LIN {X 0,Y 349.192,Z 815.635,A -85,B 0,C 180,E1 16408.843,E2 16408.843} C_VEL
LIN {X 0,Y 352.149,Z 828.309,A -85,B 0,C 180,E1 16411.517,E2 16411.517} C_VEL
LIN {X 0,Y 338.548,Z 866.043,A -85,B 0,C 180,E1 16414.618,E2 16414.618} C_VEL
LIN {X 0,Y 323.279,Z 901.225,A -85,B 0,C 180,E1 16418.786,E2 16418.786} C_VEL
LIN {X 0,Y 308.073,Z 932.384,A -85,B 0,C 180,E1 16424.048,E2 16424.048} C_VEL
LIN {X 0,Y 293.775,Z 959.9,A -85,B 0,C 180,E1 16430.633,E2 16430.633} C_VEL
LIN {X 0,Y 281.914,Z 983.359,A -85,B 0,C 180,E1 16438.716,E2 16438.716} C_VEL
LIN {X 0,Y 274.605,Z 1000.274,A -85,B 0,C 180,E1 16447.297,E2 16447.297} C_VEL
LIN {X 0,Y 271.389,Z 1010.786,A -85,B 0,C 180,E1 16455.461,E2 16455.461} C_VEL
LIN {X 0,Y 270.341,Z 1016.72,A -85,B 0,C 180,E1 16463.569,E2 16463.569} C_VEL
LIN {X 0,Y 270.547,Z 1018.167,A -85,B 0,C 180,E1 16470.001,E2 16470.001} C_VEL
LIN {X 0,Y 270.343,Z 1016.724,A -85,B 0,C 180,E1 16476.432,E2 16476.432} C_VEL
LIN {X 0,Y 271.389,Z 1010.794,A -85,B 0,C 180,E1 16484.541,E2 16484.541} C_VEL
LIN {X 0,Y 274.599,Z 1000.292,A -85,B 0,C 180,E1 16492.704,E2 16492.704} C_VEL
LIN {X 0,Y 281.856,Z 983.603,A -85,B 0,C 180,E1 16501.184,E2 16501.184} C_VEL
LIN {X 0,Y 293.699,Z 960.03,A -85,B 0,C 180,E1 16509.349,E2 16509.349} C_VEL
LIN {X 0,Y 308.953,Z 930.715,A -85,B 0,C 180,E1 16516.291,E2 16516.291} C_VEL
LIN {X 0,Y 325.073,Z 897.549,A -85,B 0,C 180,E1 16521.735,E2 16521.735} C_VEL
LIN {X 0,Y 340.684,Z 860.965,A -85,B 0,C 180,E1 16525.883,E2 16525.883} C_VEL
LIN {X 0,Y 350.17,Z 834.984,A -85,B 0,C 180,E1 16528.014,E2 16528.014} C_VEL
LIN {X 0,Y 350.059,Z 829.98,A -85,B 0,C 180,E1 16528.799,E2 16528.799} C_VEL
LIN {X 0,Y 345.076,Z 822.989,A -85,B 0,C 180,E1 16531.277,E2 16531.277} C_VEL
LIN {X 0,Y 338.35,Z 801.661,A -85,B 0,C 180,E1 16536.945,E2 16536.945} C_VEL
LIN {X 0,Y 331.725,Z 785.413,A -85,B 0,C 180,E1 16542.789,E2 16542.789} C_VEL
LIN {X 0,Y 326.179,Z 773.809,A -85,B 0,C 180,E1 16549.075,E2 16549.075} C_VEL
LIN {X 0,Y 323.36,Z 767.768,A -85,B 0,C 180,E1 16554.2,E2 16554.2} C_VEL
LIN {X 0,Y 321.912,Z 765.9,A -85,B 0,C 180,E1 16561.341,E2 16561.341} C_VEL
LIN {X 0,Y 323.589,Z 768.974,A -85,B 0,C 180,E1 16567.85,E2 16567.85} C_VEL
LIN {X 0,Y 326.59,Z 776.623,A -85,B 0,C 180,E1 16573.395,E2 16573.395} C_VEL
LIN {X 0,Y 332.226,Z 790.347,A -85,B 0,C 180,E1 16579.977,E2 16579.977} C_VEL
LIN {X 0,Y 338.405,Z 808.971,A -85,B 0,C 180,E1 16586.141,E2 16586.141} C_VEL
LIN {X 0,Y 342.983,Z 830.452,A -85,B 0,C 180,E1 16591.603,E2 16591.603} C_VEL
LIN {X 0,Y 342.674,Z 834.152,A -85,B 0,C 180,E1 16592.188,E2 16592.188} C_VEL
LIN {X 0,Y 326.849,Z 872.233,A -85,B 0,C 180,E1 16596.121,E2 16596.121} C_VEL
LIN {X 0,Y 310.06,Z 906.091,A -85,B 0,C 180,E1 16601.239,E2 16601.239} C_VEL
LIN {X 0,Y 294.191,Z 934.724,A -85,B 0,C 180,E1 16607.507,E2 16607.507} C_VEL
LIN {X 0,Y 279.881,Z 959.338,A -85,B 0,C 180,E1 16615.387,E2 16615.387} C_VEL
LIN {X 0,Y 269.909,Z 977.851,A -85,B 0,C 180,E1 16624.312,E2 16624.312} C_VEL
LIN {X 0,Y 264.694,Z 989.892,A -85,B 0,C 180,E1 16633.38,E2 16633.38} C_VEL
LIN {X 0,Y 263.017,Z 995.241,A -85,B 0,C 180,E1 16640.055,E2 16640.055} C_VEL
LIN {X 0,Y 262.515,Z 997.859,A -85,B 0,C 180,E1 16646.693,E2 16646.693} C_VEL
LIN {X 0,Y 262.472,Z 997.841,A -85,B 0,C 180,E1 16653.306,E2 16653.306} C_VEL
LIN {X 0,Y 263.46,Z 993.471,A -85,B 0,C 180,E1 16662.392,E2 16662.392} C_VEL
LIN {X 0,Y 266.708,Z 984.794,A -85,B 0,C 180,E1 16670.856,E2 16670.856} C_VEL
LIN {X 0,Y 273.935,Z 969.98,A -85,B 0,C 180,E1 16679.83,E2 16679.83} C_VEL
LIN {X 0,Y 285.315,Z 950.061,A -85,B 0,C 180,E1 16687.828,E2 16687.828} C_VEL
LIN {X 0,Y 300.025,Z 924.248,A -85,B 0,C 180,E1 16694.951,E2 16694.951} C_VEL
LIN {X 0,Y 316.458,Z 893.504,A -85,B 0,C 180,E1 16700.788,E2 16700.788} C_VEL
LIN {X 0,Y 332.912,Z 858.489,A -85,B 0,C 180,E1 16705.349,E2 16705.349} C_VEL
LIN {X 0,Y 343.162,Z 831.415,A -85,B 0,C 180,E1 16708.043,E2 16708.043} C_VEL
LIN {X 0,Y 338.289,Z 809.145,A -85,B 0,C 180,E1 16713.727,E2 16713.727} C_VEL
LIN {X 0,Y 332.65,Z 791.782,A -85,B 0,C 180,E1 16719.354,E2 16719.354} C_VEL
LIN {X 0,Y 327.088,Z 777.911,A -85,B 0,C 180,E1 16725.66,E2 16725.66} C_VEL
LIN {X 0,Y 323.78,Z 770.112,A -85,B 0,C 180,E1 16731.102,E2 16731.102} C_VEL
LIN {X 0,Y 322.787,Z 767.547,A -85,B 0,C 180,E1 16733.611,E2 16733.611} C_VEL
LIN {X 0,Y 321.875,Z 765.702,A -85,B 0,C 180,E1 16741.27,E2 16741.27} C_VEL
LIN {X 0,Y 324.017,Z 769.137,A -85,B 0,C 180,E1 16747.557,E2 16747.557} C_VEL
LIN {X 0,Y 327.173,Z 775.881,A -85,B 0,C 180,E1 16752.389,E2 16752.389} C_VEL
LIN {X 0,Y 332.03,Z 786.449,A -85,B 0,C 180,E1 16757.658,E2 16757.658} C_VEL
LIN {X 0,Y 338.631,Z 802.667,A -85,B 0,C 180,E1 16763.383,E2 16763.383} C_VEL
LIN {X 0,Y 345.418,Z 824.473,A -85,B 0,C 180,E1 16769.104,E2 16769.104} C_VEL
LIN {X 0,Y 346.743,Z 831.868,A -85,B 0,C 180,E1 16770.654,E2 16770.654} C_VEL
LIN {X 0,Y 332.245,Z 869.964,A -85,B 0,C 180,E1 16773.902,E2 16773.902} C_VEL
LIN {X 0,Y 316.574,Z 904.239,A -85,B 0,C 180,E1 16778.125,E2 16778.125} C_VEL
LIN {X 0,Y 301.211,Z 934.227,A -85,B 0,C 180,E1 16783.38,E2 16783.38} C_VEL
LIN {X 0,Y 286.56,Z 961.124,A -85,B 0,C 180,E1 16790.048,E2 16790.048} C_VEL
LIN {X 0,Y 274.435,Z 983.878,A -85,B 0,C 180,E1 16798.193,E2 16798.193} C_VEL
LIN {X 0,Y 266.586,Z 1001.235,A -85,B 0,C 180,E1 16807.458,E2 16807.458} C_VEL
LIN {X 0,Y 263.22,Z 1012.101,A -85,B 0,C 180,E1 16816.698,E2 16816.698} C_VEL
LIN {X 0,Y 262.434,Z 1016.421,A -85,B 0,C 180,E1 16823.375,E2 16823.375} C_VEL
LIN {X 0,Y 262.646,Z 1017.87,A -85,B 0,C 180,E1 16830.001,E2 16830.001} C_VEL
LIN {X 0,Y 262.437,Z 1016.426,A -85,B 0,C 180,E1 16836.627,E2 16836.627} C_VEL
LIN {X 0,Y 263.59,Z 1010.492,A -85,B 0,C 180,E1 16844.981,E2 16844.981} C_VEL
LIN {X 0,Y 267.06,Z 999.986,A -85,B 0,C 180,E1 16853.383,E2 16853.383} C_VEL
LIN {X 0,Y 275.011,Z 982.798,A -85,B 0,C 180,E1 16862.297,E2 16862.297} C_VEL
LIN {X 0,Y 287.357,Z 959.722,A -85,B 0,C 180,E1 16870.394,E2 16870.394} C_VEL
LIN {X 0,Y 302.879,Z 931.245,A -85,B 0,C 180,E1 16877.258,E2 16877.258} C_VEL
LIN {X 0,Y 319.89,Z 897.653,A -85,B 0,C 180,E1 16882.83,E2 16882.83} C_VEL
LIN {X 0,Y 335.722,Z 861.9,A -85,B 0,C 180,E1 16886.915,E2 16886.915} C_VEL
LIN {X 0,Y 346.968,Z 830.772,A -85,B 0,C 180,E1 16889.492,E2 16889.492} C_VEL
LIN {X 0,Y 345.076,Z 822.989,A -85,B 0,C 180,E1 16891.277,E2 16891.277} C_VEL
LIN {X 0,Y 341.723,Z 817.584,A -85,B 0,C 180,E1 16893.191,E2 16893.191} C_VEL
LIN {X 0,Y 335.269,Z 810.574,A -85,B 0,C 180,E1 16896.583,E2 16896.583} C_VEL
LIN {X 0,Y 329.616,Z 795.321,A -85,B 0,C 180,E1 16901.933,E2 16901.933} C_VEL
LIN {X 0,Y 324.144,Z 782.486,A -85,B 0,C 180,E1 16908.343,E2 16908.343} C_VEL
LIN {X 0,Y 320.93,Z 775.179,A -85,B 0,C 180,E1 16914.58,E2 16914.58} C_VEL
LIN {X 0,Y 319.755,Z 773.301,A -85,B 0,C 180,E1 16919.993,E2 16919.993} C_VEL
LIN {X 0,Y 320.822,Z 775.397,A -85,B 0,C 180,E1 16926.77,E2 16926.77} C_VEL
LIN {X 0,Y 324.466,Z 785.539,A -85,B 0,C 180,E1 16934.172,E2 16934.172} C_VEL
LIN {X 0,Y 329.739,Z 800.223,A -85,B 0,C 180,E1 16940.836,E2 16940.836} C_VEL
LIN {X 0,Y 334.912,Z 819.087,A -85,B 0,C 180,E1 16946.866,E2 16946.866} C_VEL
LIN {X 0,Y 337.643,Z 836.643,A -85,B 0,C 180,E1 16951.23,E2 16951.23} C_VEL
LIN {X 0,Y 321.513,Z 873.886,A -85,B 0,C 180,E1 16955.138,E2 16955.138} C_VEL
LIN {X 0,Y 304.044,Z 907.647,A -85,B 0,C 180,E1 16960.328,E2 16960.328} C_VEL
LIN {X 0,Y 287.404,Z 936.344,A -85,B 0,C 180,E1 16966.775,E2 16966.775} C_VEL
LIN {X 0,Y 273.19,Z 959.643,A -85,B 0,C 180,E1 16974.412,E2 16974.412} C_VEL
LIN {X 0,Y 262.601,Z 978.179,A -85,B 0,C 180,E1 16983.56,E2 16983.56} C_VEL
LIN {X 0,Y 257.012,Z 990.192,A -85,B 0,C 180,E1 16992.868,E2 16992.868} C_VEL
LIN {X 0,Y 255.16,Z 995.54,A -85,B 0,C 180,E1 16999.745,E2 16999.745} C_VEL
LIN {X 0,Y 254.63,Z 998.155,A -85,B 0,C 180,E1 17006.59,E2 17006.59} C_VEL
LIN {X 0,Y 254.59,Z 998.137,A -85,B 0,C 180,E1 17013.409,E2 17013.409} C_VEL
LIN {X 0,Y 255.559,Z 994.036,A -85,B 0,C 180,E1 17022.386,E2 17022.386} C_VEL
LIN {X 0,Y 259.115,Z 985.194,A -85,B 0,C 180,E1 17031.42,E2 17031.42} C_VEL
LIN {X 0,Y 266.883,Z 970.287,A -85,B 0,C 180,E1 17040.702,E2 17040.702} C_VEL
LIN {X 0,Y 279.288,Z 949.73,A -85,B 0,C 180,E1 17049.065,E2 17049.065} C_VEL
LIN {X 0,Y 294.334,Z 924.555,A -85,B 0,C 180,E1 17056.068,E2 17056.068} C_VEL
LIN {X 0,Y 311.165,Z 894.279,A -85,B 0,C 180,E1 17061.87,E2 17061.87} C_VEL
LIN {X 0,Y 327.828,Z 860.177,A -85,B 0,C 180,E1 17066.356,E2 17066.356} C_VEL
LIN {X 0,Y 337.792,Z 836.164,A -85,B 0,C 180,E1 17068.696,E2 17068.696} C_VEL
LIN {X 0,Y 334.138,Z 816.442,A -85,B 0,C 180,E1 17073.793,E2 17073.793} C_VEL
LIN {X 0,Y 328.985,Z 798.23,A -85,B 0,C 180,E1 17079.817,E2 17079.817} C_VEL
LIN {X 0,Y 323.83,Z 784.12,A -85,B 0,C 180,E1 17086.489,E2 17086.489} C_VEL
LIN {X 0,Y 320.962,Z 776.22,A -85,B 0,C 180,E1 17092.15,E2 17092.15} C_VEL
LIN {X 0,Y 319.624,Z 772.942,A -85,B 0,C 180,E1 17100.007,E2 17100.007} C_VEL
LIN {X 0,Y 321.547,Z 776.325,A -85,B 0,C 180,E1 17107.191,E2 17107.191} C_VEL
LIN {X 0,Y 326.002,Z 786.606,A -85,B 0,C 180,E1 17114.186,E2 17114.186} C_VEL
LIN {X 0,Y 332.256,Z 801.967,A -85,B 0,C 180,E1 17120.685,E2 17120.685} C_VEL
LIN {X 0,Y 338.803,Z 822.716,A -85,B 0,C 180,E1 17126.808,E2 17126.808} C_VEL
LIN {X 0,Y 341.672,Z 834.738,A -85,B 0,C 180,E1 17129.722,E2 17129.722} C_VEL
LIN {X 0,Y 325.744,Z 874.43,A -85,B 0,C 180,E1 17133.213,E2 17133.213} C_VEL
LIN {X 0,Y 308.657,Z 909.78,A -85,B 0,C 180,E1 17137.817,E2 17137.817} C_VEL
LIN {X 0,Y 291.346,Z 941.598,A -85,B 0,C 180,E1 17143.895,E2 17143.895} C_VEL
LIN {X 0,Y 275.826,Z 968.396,A -85,B 0,C 180,E1 17151.362,E2 17151.362} C_VEL
LIN {X 0,Y 264.539,Z 989.281,A -85,B 0,C 180,E1 17159.947,E2 17159.947} C_VEL
LIN {X 0,Y 257.678,Z 1004.486,A -85,B 0,C 180,E1 17169.357,E2 17169.357} C_VEL
LIN {X 0,Y 255.097,Z 1012.945,A -85,B 0,C 180,E1 17177.832,E2 17177.832} C_VEL
LIN {X 0,Y 254.608,Z 1017.208,A -85,B 0,C 180,E1 17186.591,E2 17186.591} C_VEL
LIN {X 0,Y 254.548,Z 1017.208,A -85,B 0,C 180,E1 17193.411,E2 17193.411} C_VEL
LIN {X 0,Y 255.108,Z 1012.946,A -85,B 0,C 180,E1 17202.181,E2 17202.181} C_VEL
LIN {X 0,Y 257.652,Z 1004.502,A -85,B 0,C 180,E1 17210.646,E2 17210.646} C_VEL
LIN {X 0,Y 264.538,Z 989.306,A -85,B 0,C 180,E1 17220.054,E2 17220.054} C_VEL
LIN {X 0,Y 276.522,Z 967.268,A -85,B 0,C 180,E1 17229.027,E2 17229.027} C_VEL
LIN {X 0,Y 292.299,Z 939.965,A -85,B 0,C 180,E1 17236.485,E2 17236.485} C_VEL
LIN {X 0,Y 309.624,Z 908.014,A -85,B 0,C 180,E1 17242.458,E2 17242.458} C_VEL
LIN {X 0,Y 326.654,Z 872.547,A -85,B 0,C 180,E1 17246.99,E2 17246.99} C_VEL
LIN {X 0,Y 341.581,Z 834.062,A -85,B 0,C 180,E1 17250.452,E2 17250.452} C_VEL
LIN {X 0,Y 335.818,Z 812.344,A -85,B 0,C 180,E1 17256.057,E2 17256.057} C_VEL
LIN {X 0,Y 335.269,Z 810.574,A -85,B 0,C 180,E1 17256.583,E2 17256.583} C_VEL
LIN {X 0,Y 331.982,Z 806.597,A -85,B 0,C 180,E1 17258.657,E2 17258.657} C_VEL
LIN {X 0,Y 326.134,Z 802.071,A -85,B 0,C 180,E1 17262.299,E2 17262.299} C_VEL
LIN {X 0,Y 321.4,Z 790.016,A -85,B 0,C 180,E1 17268.446,E2 17268.446} C_VEL
LIN {X 0,Y 318.386,Z 782.743,A -85,B 0,C 180,E1 17274.536,E2 17274.536} C_VEL
LIN {X 0,Y 317.226,Z 780.794,A -85,B 0,C 180,E1 17279.993,E2 17279.993} C_VEL
LIN {X 0,Y 318.241,Z 783.088,A -85,B 0,C 180,E1 17286.825,E2 17286.825} C_VEL
LIN {X 0,Y 321.541,Z 793.293,A -85,B 0,C 180,E1 17294.304,E2 17294.304} C_VEL
LIN {X 0,Y 326.297,Z 808.189,A -85,B 0,C 180,E1 17300.984,E2 17300.984} C_VEL
LIN {X 0,Y 330.606,Z 826.564,A -85,B 0,C 180,E1 17306.877,E2 17306.877} C_VEL
LIN {X 0,Y 332.243,Z 840.085,A -85,B 0,C 180,E1 17310.333,E2 17310.333} C_VEL
LIN {X 0,Y 316.498,Z 875.047,A -85,B 0,C 180,E1 17314.059,E2 17314.059} C_VEL
LIN {X 0,Y 298.871,Z 907.947,A -85,B 0,C 180,E1 17319.146,E2 17319.146} C_VEL
LIN {X 0,Y 281.49,Z 936.649,A -85,B 0,C 180,E1 17325.633,E2 17325.633} C_VEL
LIN {X 0,Y 266.334,Z 960.267,A -85,B 0,C 180,E1 17333.519,E2 17333.519} C_VEL
LIN {X 0,Y 255.33,Z 978.522,A -85,B 0,C 180,E1 17342.775,E2 17342.775} C_VEL
LIN {X 0,Y 249.319,Z 990.494,A -85,B 0,C 180,E1 17352.323,E2 17352.323} C_VEL
LIN {X 0,Y 247.312,Z 995.839,A -85,B 0,C 180,E1 17359.416,E2 17359.416} C_VEL
LIN {X 0,Y 246.725,Z 998.452,A -85,B 0,C 180,E1 17366.481,E2 17366.481} C_VEL
LIN {X 0,Y 246.685,Z 998.434,A -85,B 0,C 180,E1 17373.518,E2 17373.518} C_VEL
LIN {X 0,Y 247.568,Z 994.868,A -85,B 0,C 180,E1 17381.972,E2 17381.972} C_VEL
LIN {X 0,Y 251.095,Z 986.61,A -85,B 0,C 180,E1 17391.21,E2 17391.21} C_VEL
LIN {X 0,Y 258.948,Z 972.277,A -85,B 0,C 180,E1 17400.771,E2 17400.771} C_VEL
LIN {X 0,Y 272.273,Z 951.216,A -85,B 0,C 180,E1 17409.754,E2 17409.754} C_VEL
LIN {X 0,Y 288.749,Z 924.863,A -85,B 0,C 180,E1 17417.231,E2 17417.231} C_VEL
LIN {X 0,Y 306.107,Z 894.856,A -85,B 0,C 180,E1 17423.016,E2 17423.016} C_VEL
LIN {X 0,Y 323.791,Z 859.668,A -85,B 0,C 180,E1 17427.629,E2 17427.629} C_VEL
LIN {X 0,Y 332.434,Z 838.872,A -85,B 0,C 180,E1 17429.739,E2 17429.739} C_VEL
LIN {X 0,Y 328.718,Z 818.125,A -85,B 0,C 180,E1 17435.52,E2 17435.52} C_VEL
LIN {X 0,Y 324.28,Z 801.901,A -85,B 0,C 180,E1 17441.394,E2 17441.394} C_VEL
LIN {X 0,Y 320.216,Z 789.549,A -85,B 0,C 180,E1 17447.723,E2 17447.723} C_VEL
LIN {X 0,Y 318.024,Z 783.165,A -85,B 0,C 180,E1 17453.035,E2 17453.035} C_VEL
LIN {X 0,Y 317.101,Z 780.442,A -85,B 0,C 180,E1 17460.007,E2 17460.007} C_VEL
LIN {X 0,Y 318.933,Z 784.119,A -85,B 0,C 180,E1 17467.25,E2 17467.25} C_VEL
LIN {X 0,Y 322.662,Z 793.144,A -85,B 0,C 180,E1 17473.574,E2 17473.574} C_VEL
LIN {X 0,Y 328.407,Z 808.289,A -85,B 0,C 180,E1 17480.21,E2 17480.21} C_VEL
LIN {X 0,Y 334.045,Z 828.023,A -85,B 0,C 180,E1 17486.229,E2 17486.229} C_VEL
LIN {X 0,Y 336.04,Z 838.94,A -85,B 0,C 180,E1 17488.871,E2 17488.871} C_VEL
LIN {X 0,Y 320.665,Z 875.582,A -85,B 0,C 180,E1 17492.162,E2 17492.162} C_VEL
LIN {X 0,Y 302.655,Z 911.323,A -85,B 0,C 180,E1 17496.896,E2 17496.896} C_VEL
LIN {X 0,Y 285.213,Z 942.034,A -85,B 0,C 180,E1 17502.881,E2 17502.881} C_VEL
LIN {X 0,Y 269.365,Z 968.165,A -85,B 0,C 180,E1 17510.293,E2 17510.293} C_VEL
LIN {X 0,Y 257.431,Z 988.97,A -85,B 0,C 180,E1 17519.028,E2 17519.028} C_VEL
LIN {X 0,Y 250.048,Z 1004.179,A -85,B 0,C 180,E1 17528.697,E2 17528.697} C_VEL
LIN {X 0,Y 247.248,Z 1012.646,A -85,B 0,C 180,E1 17537.442,E2 17537.442} C_VEL
LIN {X 0,Y 246.693,Z 1016.91,A -85,B 0,C 180,E1 17546.482,E2 17546.482} C_VEL
LIN {X 0,Y 246.636,Z 1016.911,A -85,B 0,C 180,E1 17553.52,E2 17553.52} C_VEL
LIN {X 0,Y 247.241,Z 1012.764,A -85,B 0,C 180,E1 17562.406,E2 17562.406} C_VEL
LIN {X 0,Y 250.024,Z 1004.197,A -85,B 0,C 180,E1 17571.306,E2 17571.306} C_VEL
LIN {X 0,Y 257.442,Z 988.998,A -85,B 0,C 180,E1 17580.972,E2 17580.972} C_VEL
LIN {X 0,Y 270.046,Z 967.123,A -85,B 0,C 180,E1 17590.08,E2 17590.08} C_VEL
LIN {X 0,Y 286.663,Z 939.657,A -85,B 0,C 180,E1 17597.685,E2 17597.685} C_VEL
LIN {X 0,Y 304.478,Z 908.171,A -85,B 0,C 180,E1 17603.607,E2 17603.607} C_VEL
LIN {X 0,Y 322.231,Z 872.422,A -85,B 0,C 180,E1 17608.182,E2 17608.182} C_VEL
LIN {X 0,Y 336.284,Z 837.943,A -85,B 0,C 180,E1 17611.286,E2 17611.286} C_VEL
LIN {X 0,Y 331.082,Z 816.695,A -85,B 0,C 180,E1 17617.051,E2 17617.051} C_VEL
LIN {X 0,Y 326.134,Z 802.071,A -85,B 0,C 180,E1 17622.299,E2 17622.299} C_VEL
LIN {X 0,Y 323.169,Z 799.664,A -85,B 0,C 180,E1 17624.521,E2 17624.521} C_VEL
LIN {X 0,Y 318.665,Z 798.307,A -85,B 0,C 180,E1 17627.991,E2 17627.991} C_VEL
LIN {X 0,Y 318.417,Z 797.734,A -85,B 0,C 180,E1 17628.374,E2 17628.374} C_VEL
LIN {X 0,Y 315.746,Z 790.323,A -85,B 0,C 180,E1 17634.491,E2 17634.491} C_VEL
LIN {X 0,Y 314.656,Z 788.271,A -85,B 0,C 180,E1 17639.993,E2 17639.993} C_VEL
LIN {X 0,Y 315.442,Z 790.714,A -85,B 0,C 180,E1 17646.884,E2 17646.884} C_VEL
LIN {X 0,Y 318.445,Z 801.039,A -85,B 0,C 180,E1 17654.408,E2 17654.408} C_VEL
LIN {X 0,Y 322.289,Z 814.685,A -85,B 0,C 180,E1 17660.619,E2 17660.619} C_VEL
LIN {X 0,Y 325.89,Z 832.625,A -85,B 0,C 180,E1 17666.516,E2 17666.516} C_VEL
LIN {X 0,Y 327.024,Z 843.334,A -85,B 0,C 180,E1 17669.394,E2 17669.394} C_VEL
LIN {X 0,Y 310.953,Z 877.44,A -85,B 0,C 180,E1 17673.109,E2 17673.109} C_VEL
LIN {X 0,Y 293.385,Z 908.928,A -85,B 0,C 180,E1 17678.047,E2 17678.047} C_VEL
LIN {X 0,Y 275.757,Z 936.95,A -85,B 0,C 180,E1 17684.456,E2 17684.456} C_VEL
LIN {X 0,Y 259.6,Z 960.887,A -85,B 0,C 180,E1 17692.587,E2 17692.587} C_VEL
LIN {X 0,Y 248.467,Z 978.3,A -85,B 0,C 180,E1 17701.556,E2 17701.556} C_VEL
LIN {X 0,Y 241.674,Z 990.794,A -85,B 0,C 180,E1 17711.744,E2 17711.744} C_VEL
LIN {X 0,Y 239.503,Z 996.137,A -85,B 0,C 180,E1 17719.067,E2 17719.067} C_VEL
LIN {X 0,Y 238.819,Z 998.749,A -85,B 0,C 180,E1 17726.364,E2 17726.364} C_VEL
LIN {X 0,Y 238.78,Z 998.731,A -85,B 0,C 180,E1 17733.635,E2 17733.635} C_VEL
LIN {X 0,Y 239.749,Z 995.168,A -85,B 0,C 180,E1 17742.369,E2 17742.369} C_VEL
LIN {X 0,Y 243.563,Z 986.915,A -85,B 0,C 180,E1 17751.899,E2 17751.899} C_VEL
LIN {X 0,Y 251.96,Z 972.585,A -85,B 0,C 180,E1 17761.722,E2 17761.722} C_VEL
LIN {X 0,Y 266.018,Z 951.526,A -85,B 0,C 180,E1 17770.884,E2 17770.884} C_VEL
LIN {X 0,Y 283.284,Z 925.172,A -85,B 0,C 180,E1 17778.44,E2 17778.44} C_VEL
LIN {X 0,Y 301.613,Z 894.615,A -85,B 0,C 180,E1 17784.328,E2 17784.328} C_VEL
LIN {X 0,Y 319.425,Z 860.312,A -85,B 0,C 180,E1 17788.806,E2 17788.806} C_VEL
LIN {X 0,Y 327.031,Z 842.333,A -85,B 0,C 180,E1 17790.694,E2 17790.694} C_VEL
LIN {X 0,Y 323.919,Z 822.212,A -85,B 0,C 180,E1 17796.6,E2 17796.6} C_VEL
LIN {X 0,Y 320.013,Z 806.768,A -85,B 0,C 180,E1 17802.563,E2 17802.563} C_VEL
LIN {X 0,Y 316.592,Z 795.336,A -85,B 0,C 180,E1 17808.98,E2 17808.98} C_VEL
LIN {X 0,Y 314.85,Z 789.72,A -85,B 0,C 180,E1 17814.488,E2 17814.488} C_VEL
LIN {X 0,Y 314.55,Z 787.914,A -85,B 0,C 180,E1 17820.007,E2 17820.007} C_VEL
LIN {X 0,Y 316.081,Z 791.293,A -85,B 0,C 180,E1 17826.884,E2 17826.884} C_VEL
LIN {X 0,Y 319.714,Z 800.938,A -85,B 0,C 180,E1 17833.702,E2 17833.702} C_VEL
LIN {X 0,Y 324.614,Z 815.273,A -85,B 0,C 180,E1 17839.99,E2 17839.99} C_VEL
LIN {X 0,Y 329.514,Z 834.289,A -85,B 0,C 180,E1 17845.885,E2 17845.885} C_VEL
LIN {X 0,Y 330.722,Z 842.44,A -85,B 0,C 180,E1 17847.94,E2 17847.94} C_VEL
LIN {X 0,Y 314.941,Z 878.272,A -85,B 0,C 180,E1 17851.254,E2 17851.254} C_VEL
LIN {X 0,Y 297.03,Z 912.353,A -85,B 0,C 180,E1 17855.857,E2 17855.857} C_VEL
LIN {X 0,Y 279.127,Z 942.546,A -85,B 0,C 180,E1 17861.842,E2 17861.842} C_VEL
LIN {X 0,Y 263.218,Z 967.625,A -85,B 0,C 180,E1 17869.061,E2 17869.061} C_VEL
LIN {X 0,Y 249.941,Z 989.378,A -85,B 0,C 180,E1 17878.455,E2 17878.455} C_VEL
LIN {X 0,Y 242.482,Z 1003.873,A -85,B 0,C 180,E1 17887.998,E2 17887.998} C_VEL
LIN {X 0,Y 239.379,Z 1012.472,A -85,B 0,C 180,E1 17897.211,E2 17897.211} C_VEL
LIN {X 0,Y 238.777,Z 1016.613,A -85,B 0,C 180,E1 17906.365,E2 17906.365} C_VEL
LIN {X 0,Y 238.997,Z 1016.983,A -85,B 0,C 180,E1 17910.001,E2 17910.001} C_VEL
LIN {X 0,Y 238.774,Z 1015.533,A -85,B 0,C 180,E1 17917.287,E2 17917.287} C_VEL
LIN {X 0,Y 240.244,Z 1009.585,A -85,B 0,C 180,E1 17926.476,E2 17926.476} C_VEL
LIN {X 0,Y 245.178,Z 998.055,A -85,B 0,C 180,E1 17936.336,E2 17936.336} C_VEL
LIN {X 0,Y 254.591,Z 981.512,A -85,B 0,C 180,E1 17945.44,E2 17945.44} C_VEL
LIN {X 0,Y 269.509,Z 957.981,A -85,B 0,C 180,E1 17954.046,E2 17954.046} C_VEL
LIN {X 0,Y 286.972,Z 929.845,A -85,B 0,C 180,E1 17960.979,E2 17960.979} C_VEL
LIN {X 0,Y 305.496,Z 897.168,A -85,B 0,C 180,E1 17966.435,E2 17966.435} C_VEL
LIN {X 0,Y 323.506,Z 860.096,A -85,B 0,C 180,E1 17970.603,E2 17970.603} C_VEL
LIN {X 0,Y 330.943,Z 841.734,A -85,B 0,C 180,E1 17972.176,E2 17972.176} C_VEL
LIN {X 0,Y 326.758,Z 822.529,A -85,B 0,C 180,E1 17977.594,E2 17977.594} C_VEL
LIN {X 0,Y 321.803,Z 806.64,A -85,B 0,C 180,E1 17983.598,E2 17983.598} C_VEL
LIN {X 0,Y 318.417,Z 797.734,A -85,B 0,C 180,E1 17988.374,E2 17988.374} C_VEL
LIN {X 0,Y 316.353,Z 796.484,A -85,B 0,C 180,E1 17990.69,E2 17990.69} C_VEL
LIN {X 0,Y 312.754,Z 797.678,A -85,B 0,C 180,E1 17994.678,E2 17994.678} C_VEL
LIN {X 0,Y 311.787,Z 795.642,A -85,B 0,C 180,E1 17999.993,E2 17999.993} C_VEL
LIN {X 0,Y 312.513,Z 798.292,A -85,B 0,C 180,E1 18006.949,E2 18006.949} C_VEL
LIN {X 0,Y 314.834,Z 807.547,A -85,B 0,C 180,E1 18013.905,E2 18013.905} C_VEL
LIN {X 0,Y 318.27,Z 821.612,A -85,B 0,C 180,E1 18020.435,E2 18020.435} C_VEL
LIN {X 0,Y 321.02,Z 837.659,A -85,B 0,C 180,E1 18025.855,E2 18025.855} C_VEL
LIN {X 0,Y 321.768,Z 846.913,A -85,B 0,C 180,E1 18028.46,E2 18028.46} C_VEL
LIN {X 0,Y 303.775,Z 883.088,A -85,B 0,C 180,E1 18032.566,E2 18032.566} C_VEL
LIN {X 0,Y 285.136,Z 914.538,A -85,B 0,C 180,E1 18037.826,E2 18037.826} C_VEL
LIN {X 0,Y 267.542,Z 940.913,A -85,B 0,C 180,E1 18044.29,E2 18044.29} C_VEL
LIN {X 0,Y 251.815,Z 963.069,A -85,B 0,C 180,E1 18052.301,E2 18052.301} C_VEL
LIN {X 0,Y 240.86,Z 979.29,A -85,B 0,C 180,E1 18061.117,E2 18061.117} C_VEL
LIN {X 0,Y 234.028,Z 991.096,A -85,B 0,C 180,E1 18071.126,E2 18071.126} C_VEL
LIN {X 0,Y 231.664,Z 996.436,A -85,B 0,C 180,E1 18078.692,E2 18078.692} C_VEL
LIN {X 0,Y 230.914,Z 999.046,A -85,B 0,C 180,E1 18086.24,E2 18086.24} C_VEL
LIN {X 0,Y 230.875,Z 999.029,A -85,B 0,C 180,E1 18093.759,E2 18093.759} C_VEL
LIN {X 0,Y 232.041,Z 995.219,A -85,B 0,C 180,E1 18103.199,E2 18103.199} C_VEL
LIN {X 0,Y 236.06,Z 987.22,A -85,B 0,C 180,E1 18112.633,E2 18112.633} C_VEL
LIN {X 0,Y 245.081,Z 972.891,A -85,B 0,C 180,E1 18122.721,E2 18122.721} C_VEL
LIN {X 0,Y 259.881,Z 951.835,A -85,B 0,C 180,E1 18132.066,E2 18132.066} C_VEL
LIN {X 0,Y 277.974,Z 925.478,A -85,B 0,C 180,E1 18139.689,E2 18139.689} C_VEL
LIN {X 0,Y 296.701,Z 895.391,A -85,B 0,C 180,E1 18145.525,E2 18145.525} C_VEL
LIN {X 0,Y 315.527,Z 860.249,A -85,B 0,C 180,E1 18150.087,E2 18150.087} C_VEL
LIN {X 0,Y 321.778,Z 846.533,A -85,B 0,C 180,E1 18151.484,E2 18151.484} C_VEL
LIN {X 0,Y 319.361,Z 827.786,A -85,B 0,C 180,E1 18157.197,E2 18157.197} C_VEL
LIN {X 0,Y 316.073,Z 812.545,A -85,B 0,C 180,E1 18163.346,E2 18163.346} C_VEL
LIN {X 0,Y 313.505,Z 802.924,A -85,B 0,C 180,E1 18168.87,E2 18168.87} C_VEL
LIN {X 0,Y 311.981,Z 797.125,A -85,B 0,C 180,E1 18174.437,E2 18174.437} C_VEL
LIN {X 0,Y 311.69,Z 795.265,A -85,B 0,C 180,E1 18180.007,E2 18180.007} C_VEL
LIN {X 0,Y 313.153,Z 798.871,A -85,B 0,C 180,E1 18186.948,E2 18186.948} C_VEL
LIN {X 0,Y 316.552,Z 808.715,A -85,B 0,C 180,E1 18193.841,E2 18193.841} C_VEL
LIN {X 0,Y 321.024,Z 823.438,A -85,B 0,C 180,E1 18200.223,E2 18200.223} C_VEL
LIN {X 0,Y 325.257,Z 843.257,A -85,B 0,C 180,E1 18206.338,E2 18206.338} C_VEL
LIN {X 0,Y 325.147,Z 846.868,A -85,B 0,C 180,E1 18207.056,E2 18207.056} C_VEL
LIN {X 0,Y 307.223,Z 885.137,A -85,B 0,C 180,E1 18210.789,E2 18210.789} C_VEL
LIN {X 0,Y 287.573,Z 920.096,A -85,B 0,C 180,E1 18215.921,E2 18215.921} C_VEL
LIN {X 0,Y 268.015,Z 950.844,A -85,B 0,C 180,E1 18222.744,E2 18222.744} C_VEL
LIN {X 0,Y 252.275,Z 974.556,A -85,B 0,C 180,E1 18230.6,E2 18230.6} C_VEL
LIN {X 0,Y 239.665,Z 994.572,A -85,B 0,C 180,E1 18240.669,E2 18240.669} C_VEL
LIN {X 0,Y 233.183,Z 1007.612,A -85,B 0,C 180,E1 18251.056,E2 18251.056} C_VEL
LIN {X 0,Y 231.216,Z 1013.684,A -85,B 0,C 180,E1 18259.196,E2 18259.196} C_VEL
LIN {X 0,Y 230.862,Z 1016.315,A -85,B 0,C 180,E1 18266.24,E2 18266.24} C_VEL
LIN {X 0,Y 231.094,Z 1016.687,A -85,B 0,C 180,E1 18270.001,E2 18270.001} C_VEL
LIN {X 0,Y 230.87,Z 1015.234,A -85,B 0,C 180,E1 18277.538,E2 18277.538} C_VEL
LIN {X 0,Y 232.504,Z 1009.282,A -85,B 0,C 180,E1 18287.041,E2 18287.041} C_VEL
LIN {X 0,Y 237.564,Z 998.303,A -85,B 0,C 180,E1 18296.836,E2 18296.836} C_VEL
LIN {X 0,Y 247.91,Z 981.204,A -85,B 0,C 180,E1 18306.547,E2 18306.547} C_VEL
LIN {X 0,Y 263.579,Z 957.67,A -85,B 0,C 180,E1 18315.306,E2 18315.306} C_VEL
LIN {X 0,Y 282.245,Z 928.954,A -85,B 0,C 180,E1 18322.386,E2 18322.386} C_VEL
LIN {X 0,Y 301.71,Z 895.704,A -85,B 0,C 180,E1 18327.871,E2 18327.871} C_VEL
LIN {X 0,Y 319.57,Z 859.865,A -85,B 0,C 180,E1 18331.865,E2 18331.865} C_VEL
LIN {X 0,Y 325.572,Z 844.966,A -85,B 0,C 180,E1 18333.248,E2 18333.248} C_VEL
LIN {X 0,Y 321.509,Z 824.984,A -85,B 0,C 180,E1 18339.259,E2 18339.259} C_VEL
LIN {X 0,Y 317.068,Z 810.228,A -85,B 0,C 180,E1 18345.476,E2 18345.476} C_VEL
LIN {X 0,Y 313.68,Z 800.94,A -85,B 0,C 180,E1 18351.668,E2 18351.668} C_VEL
LIN {X 0,Y 312.754,Z 797.678,A -85,B 0,C 180,E1 18354.678,E2 18354.678} C_VEL
LIN {X 0,Y 310.524,Z 799.884,A -85,B 0,C 180,E1 18357.834,E2 18357.834} C_VEL
LIN {X 0,Y 308.724,Z 803.184,A -85,B 0,C 180,E1 18361.031,E2 18361.031} C_VEL
LIN {X 0,Y 309.335,Z 805.751,A -85,B 0,C 180,E1 18367.021,E2 18367.021} C_VEL
LIN {X 0,Y 311.402,Z 815.214,A -85,B 0,C 180,E1 18374.061,E2 18374.061} C_VEL
LIN {X 0,Y 314.185,Z 828.907,A -85,B 0,C 180,E1 18380.44,E2 18380.44} C_VEL
LIN {X 0,Y 316.173,Z 844.803,A -85,B 0,C 180,E1 18385.851,E2 18385.851} C_VEL
LIN {X 0,Y 316.266,Z 851.098,A -85,B 0,C 180,E1 18387.563,E2 18387.563} C_VEL
LIN {X 0,Y 298.116,Z 885.934,A -85,B 0,C 180,E1 18391.615,E2 18391.615} C_VEL
LIN {X 0,Y 278.627,Z 917.35,A -85,B 0,C 180,E1 18397.018,E2 18397.018} C_VEL
LIN {X 0,Y 259.555,Z 944.57,A -85,B 0,C 180,E1 18404.024,E2 18404.024} C_VEL
LIN {X 0,Y 243.16,Z 966.57,A -85,B 0,C 180,E1 18412.62,E2 18412.62} C_VEL
LIN {X 0,Y 231.364,Z 983.142,A -85,B 0,C 180,E1 18422.735,E2 18422.735} C_VEL
LIN {X 0,Y 225.569,Z 992.917,A -85,B 0,C 180,E1 18432.418,E2 18432.418} C_VEL
LIN {X 0,Y 223.185,Z 998.374,A -85,B 0,C 180,E1 18442.201,E2 18442.201} C_VEL
LIN {X 0,Y 223.148,Z 999.652,A -85,B 0,C 180,E1 18449.999,E2 18449.999} C_VEL
LIN {X 0,Y 223.157,Z 998.338,A -85,B 0,C 180,E1 18457.798,E2 18457.798} C_VEL
LIN {X 0,Y 225.585,Z 992.833,A -85,B 0,C 180,E1 18467.579,E2 18467.579} C_VEL
LIN {X 0,Y 231.411,Z 982.998,A -85,B 0,C 180,E1 18477.257,E2 18477.257} C_VEL
LIN {X 0,Y 243.259,Z 966.37,A -85,B 0,C 180,E1 18487.36,E2 18487.36} C_VEL
LIN {X 0,Y 260.061,Z 943.735,A -85,B 0,C 180,E1 18496.12,E2 18496.12} C_VEL
LIN {X 0,Y 279.032,Z 916.571,A -85,B 0,C 180,E1 18503.031,E2 18503.031} C_VEL
LIN {X 0,Y 298.454,Z 885.205,A -85,B 0,C 180,E1 18508.37,E2 18508.37} C_VEL
LIN {X 0,Y 316.482,Z 849.634,A -85,B 0,C 180,E1 18512.614,E2 18512.614} C_VEL
LIN {X 0,Y 314.353,Z 830.435,A -85,B 0,C 180,E1 18518.834,E2 18518.834} C_VEL
LIN {X 0,Y 311.505,Z 816.208,A -85,B 0,C 180,E1 18525.224,E2 18525.224} C_VEL
LIN {X 0,Y 309.401,Z 807.017,A -85,B 0,C 180,E1 18531.566,E2 18531.566} C_VEL
LIN {X 0,Y 308.597,Z 803.269,A -85,B 0,C 180,E1 18537.195,E2 18537.195} C_VEL
LIN {X 0,Y 308.776,Z 802.609,A -85,B 0,C 180,E1 18540.007,E2 18540.007} C_VEL
LIN {X 0,Y 309.969,Z 805.876,A -85,B 0,C 180,E1 18546.572,E2 18546.572} C_VEL
LIN {X 0,Y 312.87,Z 815.151,A -85,B 0,C 180,E1 18553.321,E2 18553.321} C_VEL
LIN {X 0,Y 316.631,Z 829.026,A -85,B 0,C 180,E1 18559.56,E2 18559.56} C_VEL
LIN {X 0,Y 320.153,Z 847.535,A -85,B 0,C 180,E1 18565.499,E2 18565.499} C_VEL
LIN {X 0,Y 319.427,Z 851.382,A -85,B 0,C 180,E1 18566.173,E2 18566.173} C_VEL
LIN {X 0,Y 301.882,Z 887.105,A -85,B 0,C 180,E1 18569.742,E2 18569.742} C_VEL
LIN {X 0,Y 282.415,Z 920.432,A -85,B 0,C 180,E1 18574.694,E2 18574.694} C_VEL
LIN {X 0,Y 262.512,Z 950.534,A -85,B 0,C 180,E1 18581.428,E2 18581.428} C_VEL
LIN {X 0,Y 245.461,Z 974.863,A -85,B 0,C 180,E1 18589.634,E2 18589.634} C_VEL
LIN {X 0,Y 232.506,Z 994.284,A -85,B 0,C 180,E1 18599.691,E2 18599.691} C_VEL
LIN {X 0,Y 225.498,Z 1007.306,A -85,B 0,C 180,E1 18610.384,E2 18610.384} C_VEL
LIN {X 0,Y 223.409,Z 1013.123,A -85,B 0,C 180,E1 18618.27,E2 18618.27} C_VEL
LIN {X 0,Y 222.967,Z 1016.018,A -85,B 0,C 180,E1 18626.107,E2 18626.107} C_VEL
LIN {X 0,Y 223.19,Z 1016.391,A -85,B 0,C 180,E1 18630.001,E2 18630.001} C_VEL
LIN {X 0,Y 222.981,Z 1014.936,A -85,B 0,C 180,E1 18637.806,E2 18637.806} C_VEL
LIN {X 0,Y 224.773,Z 1008.979,A -85,B 0,C 180,E1 18647.646,E2 18647.646} C_VEL
LIN {X 0,Y 229.991,Z 998.453,A -85,B 0,C 180,E1 18657.441,E2 18657.441} C_VEL
LIN {X 0,Y 241.331,Z 980.896,A -85,B 0,C 180,E1 18667.714,E2 18667.714} C_VEL
LIN {X 0,Y 257.751,Z 957.458,A -85,B 0,C 180,E1 18676.587,E2 18676.587} C_VEL
LIN {X 0,Y 276.759,Z 929.538,A -85,B 0,C 180,E1 18683.555,E2 18683.555} C_VEL
LIN {X 0,Y 297.127,Z 896.004,A -85,B 0,C 180,E1 18689.123,E2 18689.123} C_VEL
LIN {X 0,Y 315.822,Z 859.599,A -85,B 0,C 180,E1 18693.156,E2 18693.156} C_VEL
LIN {X 0,Y 320.355,Z 848.66,A -85,B 0,C 180,E1 18694.213,E2 18694.213} C_VEL
LIN {X 0,Y 317.203,Z 831.018,A -85,B 0,C 180,E1 18699.749,E2 18699.749} C_VEL
LIN {X 0,Y 313.334,Z 816.625,A -85,B 0,C 180,E1 18706.014,E2 18706.014} C_VEL
LIN {X 0,Y 310.545,Z 808.382,A -85,B 0,C 180,E1 18711.584,E2 18711.584} C_VEL
LIN {X 0,Y 309.684,Z 805.046,A -85,B 0,C 180,E1 18714.774,E2 18714.774} C_VEL
LIN {X 0,Y 308.724,Z 803.184,A -85,B 0,C 180,E1 18721.031,E2 18721.031} C_VEL
LIN {X 0,Y 307.794,Z 805.979,A -85,B 0,C 180,E1 18723.401,E2 18723.401} C_VEL
LIN {X 0,Y 306.081,Z 813.398,A -85,B 0,C 180,E1 18727.287,E2 18727.287} C_VEL
LIN {X 0,Y 307.496,Z 821.402,A -85,B 0,C 180,E1 18733.445,E2 18733.445} C_VEL
LIN {X 0,Y 309.628,Z 833.858,A -85,B 0,C 180,E1 18739.549,E2 18739.549} C_VEL
LIN {X 0,Y 311.218,Z 850.267,A -85,B 0,C 180,E1 18745.346,E2 18745.346} C_VEL
LIN {X 0,Y 310.764,Z 855.145,A -85,B 0,C 180,E1 18746.631,E2 18746.631} C_VEL
LIN {X 0,Y 292.849,Z 888.044,A -85,B 0,C 180,E1 18750.539,E2 18750.539} C_VEL
LIN {X 0,Y 272.185,Z 919.934,A -85,B 0,C 180,E1 18756.159,E2 18756.159} C_VEL
LIN {X 0,Y 253.386,Z 945.623,A -85,B 0,C 180,E1 18762.946,E2 18762.946} C_VEL
LIN {X 0,Y 236.693,Z 966.874,A -85,B 0,C 180,E1 18771.413,E2 18771.413} C_VEL
LIN {X 0,Y 224.185,Z 983.445,A -85,B 0,C 180,E1 18781.786,E2 18781.786} C_VEL
LIN {X 0,Y 217.905,Z 993.218,A -85,B 0,C 180,E1 18791.779,E2 18791.779} C_VEL
LIN {X 0,Y 215.309,Z 998.672,A -85,B 0,C 180,E1 18801.914,E2 18801.914} C_VEL
LIN {X 0,Y 215.247,Z 999.949,A -85,B 0,C 180,E1 18809.999,E2 18809.999} C_VEL
LIN {X 0,Y 215.692,Z 997.554,A -85,B 0,C 180,E1 18820.752,E2 18820.752} C_VEL
LIN {X 0,Y 218.853,Z 991.599,A -85,B 0,C 180,E1 18830.237,E2 18830.237} C_VEL
LIN {X 0,Y 227.184,Z 979.265,A -85,B 0,C 180,E1 18841.225,E2 18841.225} C_VEL
LIN {X 0,Y 241.364,Z 960.974,A -85,B 0,C 180,E1 18851.192,E2 18851.192} C_VEL
LIN {X 0,Y 260.251,Z 936.407,A -85,B 0,C 180,E1 18859.712,E2 18859.712} C_VEL
LIN {X 0,Y 280.292,Z 907.888,A -85,B 0,C 180,E1 18866.152,E2 18866.152} C_VEL
LIN {X 0,Y 301.143,Z 873.495,A -85,B 0,C 180,E1 18871.258,E2 18871.258} C_VEL
LIN {X 0,Y 310.809,Z 854.783,A -85,B 0,C 180,E1 18873.302,E2 18873.302} C_VEL
LIN {X 0,Y 310.383,Z 841.273,A -85,B 0,C 180,E1 18877.524,E2 18877.524} C_VEL
LIN {X 0,Y 308.372,Z 826.596,A -85,B 0,C 180,E1 18883.611,E2 18883.611} C_VEL
LIN {X 0,Y 306.533,Z 816.796,A -85,B 0,C 180,E1 18889.455,E2 18889.455} C_VEL
LIN {X 0,Y 305.702,Z 811.787,A -85,B 0,C 180,E1 18894.323,E2 18894.323} C_VEL
LIN {X 0,Y 305.575,Z 809.847,A -85,B 0,C 180,E1 18900.007,E2 18900.007} C_VEL
LIN {X 0,Y 306.712,Z 813.263,A -85,B 0,C 180,E1 18906.626,E2 18906.626} C_VEL
LIN {X 0,Y 309.356,Z 822.743,A -85,B 0,C 180,E1 18913.476,E2 18913.476} C_VEL
LIN {X 0,Y 312.663,Z 837.025,A -85,B 0,C 180,E1 18919.819,E2 18919.819} C_VEL
LIN {X 0,Y 315.025,Z 852.465,A -85,B 0,C 180,E1 18924.871,E2 18924.871} C_VEL
LIN {X 0,Y 297.264,Z 887.951,A -85,B 0,C 180,E1 18928.526,E2 18928.526} C_VEL
LIN {X 0,Y 277.169,Z 921.08,A -85,B 0,C 180,E1 18933.48,E2 18933.48} C_VEL
LIN {X 0,Y 257.105,Z 950.221,A -85,B 0,C 180,E1 18940.044,E2 18940.044} C_VEL
LIN {X 0,Y 239.193,Z 974.55,A -85,B 0,C 180,E1 18948.346,E2 18948.346} C_VEL
LIN {X 0,Y 225.428,Z 993.974,A -85,B 0,C 180,E1 18958.633,E2 18958.633} C_VEL
LIN {X 0,Y 217.866,Z 1007.001,A -85,B 0,C 180,E1 18969.668,E2 18969.668} C_VEL
LIN {X 0,Y 215.175,Z 1013.843,A -85,B 0,C 180,E1 18980.113,E2 18980.113} C_VEL
LIN {X 0,Y 215.285,Z 1016.094,A -85,B 0,C 180,E1 18990.001,E2 18990.001} C_VEL
LIN {X 0,Y 215.18,Z 1013.849,A -85,B 0,C 180,E1 18999.895,E2 18999.895} C_VEL
LIN {X 0,Y 217.848,Z 1007.02,A -85,B 0,C 180,E1 19010.336,E2 19010.336} C_VEL
LIN {X 0,Y 225.425,Z 994.007,A -85,B 0,C 180,E1 19021.369,E2 19021.369} C_VEL
LIN {X 0,Y 239.182,Z 974.595,A -85,B 0,C 180,E1 19031.659,E2 19031.659} C_VEL
LIN {X 0,Y 258.171,Z 948.927,A -85,B 0,C 180,E1 19040.331,E2 19040.331} C_VEL
LIN {X 0,Y 279.067,Z 918.371,A -85,B 0,C 180,E1 19047.021,E2 19047.021} C_VEL
LIN {X 0,Y 299.997,Z 883.297,A -85,B 0,C 180,E1 19052.035,E2 19052.035} C_VEL
LIN {X 0,Y 314.85,Z 853.695,A -85,B 0,C 180,E1 19054.942,E2 19054.942} C_VEL
LIN {X 0,Y 313.218,Z 839.573,A -85,B 0,C 180,E1 19059.294,E2 19059.294} C_VEL
LIN {X 0,Y 310.172,Z 825.66,A -85,B 0,C 180,E1 19065.08,E2 19065.08} C_VEL
LIN {X 0,Y 307.31,Z 815.776,A -85,B 0,C 180,E1 19071.494,E2 19071.494} C_VEL
LIN {X 0,Y 306.59,Z 812.603,A -85,B 0,C 180,E1 19074.326,E2 19074.326} C_VEL
LIN {X 0,Y 305.532,Z 810.398,A -85,B 0,C 180,E1 19080.973,E2 19080.973} C_VEL
LIN {X 0,Y 306.072,Z 813.184,A -85,B 0,C 180,E1 19087.096,E2 19087.096} C_VEL
LIN {X 0,Y 306.081,Z 813.398,A -85,B 0,C 180,E1 19087.287,E2 19087.287} C_VEL
LIN {X 0,Y 304.801,Z 820.426,A -85,B 0,C 180,E1 19090.287,E2 19090.287} C_VEL
LIN {X 0,Y 303.651,Z 828.328,A -85,B 0,C 180,E1 19093.271,E2 19093.271} C_VEL
LIN {X 0,Y 305.268,Z 841.014,A -85,B 0,C 180,E1 19099.544,E2 19099.544} C_VEL
LIN {X 0,Y 306.062,Z 855.728,A -85,B 0,C 180,E1 19104.877,E2 19104.877} C_VEL
LIN {X 0,Y 305.41,Z 859.09,A -85,B 0,C 180,E1 19105.662,E2 19105.662} C_VEL
LIN {X 0,Y 286.379,Z 892.204,A -85,B 0,C 180,E1 19109.721,E2 19109.721} C_VEL
LIN {X 0,Y 266.087,Z 922.114,A -85,B 0,C 180,E1 19115.174,E2 19115.174} C_VEL
LIN {X 0,Y 246.914,Z 947.105,A -85,B 0,C 180,E1 19121.968,E2 19121.968} C_VEL
LIN {X 0,Y 228.927,Z 968.92,A -85,B 0,C 180,E1 19131.073,E2 19131.073} C_VEL
LIN {X 0,Y 216.147,Z 984.927,A -85,B 0,C 180,E1 19141.781,E2 19141.781} C_VEL
LIN {X 0,Y 209.437,Z 995.018,A -85,B 0,C 180,E1 19153.191,E2 19153.191} C_VEL
LIN {X 0,Y 207.459,Z 998.969,A -85,B 0,C 180,E1 19161.606,E2 19161.606} C_VEL
LIN {X 0,Y 207.358,Z 1000.244,A -85,B 0,C 180,E1 19169.999,E2 19169.999} C_VEL
LIN {X 0,Y 207.435,Z 998.934,A -85,B 0,C 180,E1 19178.393,E2 19178.393} C_VEL
LIN {X 0,Y 210.281,Z 993.438,A -85,B 0,C 180,E1 19188.905,E2 19188.905} C_VEL
LIN {X 0,Y 217.835,Z 982.611,A -85,B 0,C 180,E1 19199.994,E2 19199.994} C_VEL
LIN {X 0,Y 230.47,Z 966.985,A -85,B 0,C 180,E1 19209.83,E2 19209.83} C_VEL
LIN {X 0,Y 248.984,Z 944.41,A -85,B 0,C 180,E1 19218.809,E2 19218.809} C_VEL
LIN {X 0,Y 270.039,Z 916.544,A -85,B 0,C 180,E1 19225.911,E2 19225.911} C_VEL
LIN {X 0,Y 290.636,Z 885.296,A -85,B 0,C 180,E1 19231.145,E2 19231.145} C_VEL
LIN {X 0,Y 305.997,Z 857.403,A -85,B 0,C 180,E1 19234.457,E2 19234.457} C_VEL
LIN {X 0,Y 305.146,Z 840.51,A -85,B 0,C 180,E1 19240.517,E2 19240.517} C_VEL
LIN {X 0,Y 303.459,Z 827.536,A -85,B 0,C 180,E1 19247.034,E2 19247.034} C_VEL
LIN {X 0,Y 302.276,Z 818.986,A -85,B 0,C 180,E1 19254.258,E2 19254.258} C_VEL
LIN {X 0,Y 302.299,Z 817.051,A -85,B 0,C 180,E1 19260.007,E2 19260.007} C_VEL
LIN {X 0,Y 303.282,Z 820.592,A -85,B 0,C 180,E1 19266.701,E2 19266.701} C_VEL
LIN {X 0,Y 305.37,Z 828.97,A -85,B 0,C 180,E1 19272.897,E2 19272.897} C_VEL
LIN {X 0,Y 308.174,Z 843.003,A -85,B 0,C 180,E1 19279.364,E2 19279.364} C_VEL
LIN {X 0,Y 309.686,Z 857.022,A -85,B 0,C 180,E1 19284.028,E2 19284.028} C_VEL
LIN {X 0,Y 290.748,Z 892.302,A -85,B 0,C 180,E1 19287.715,E2 19287.715} C_VEL
LIN {X 0,Y 271.169,Z 923,A -85,B 0,C 180,E1 19292.459,E2 19292.459} C_VEL
LIN {X 0,Y 250.65,Z 951.47,A -85,B 0,C 180,E1 19299.054,E2 19299.054} C_VEL
LIN {X 0,Y 232.248,Z 975.236,A -85,B 0,C 180,E1 19307.44,E2 19307.44} C_VEL
LIN {X 0,Y 218.432,Z 993.664,A -85,B 0,C 180,E1 19317.508,E2 19317.508} C_VEL
LIN {X 0,Y 210.245,Z 1006.695,A -85,B 0,C 180,E1 19328.896,E2 19328.896} C_VEL
LIN {X 0,Y 207.732,Z 1012.521,A -85,B 0,C 180,E1 19337.371,E2 19337.371} C_VEL
LIN {X 0,Y 207.158,Z 1015.424,A -85,B 0,C 180,E1 19345.809,E2 19345.809} C_VEL
LIN {X 0,Y 207.396,Z 1015.798,A -85,B 0,C 180,E1 19350.001,E2 19350.001} C_VEL
LIN {X 0,Y 207.2,Z 1014.339,A -85,B 0,C 180,E1 19358.405,E2 19358.405} C_VEL
LIN {X 0,Y 209.239,Z 1008.684,A -85,B 0,C 180,E1 19368.586,E2 19368.586} C_VEL
LIN {X 0,Y 215.531,Z 997.838,A -85,B 0,C 180,E1 19379.456,E2 19379.456} C_VEL
LIN {X 0,Y 228.266,Z 980.553,A -85,B 0,C 180,E1 19390.124,E2 19390.124} C_VEL
LIN {X 0,Y 246.618,Z 956.901,A -85,B 0,C 180,E1 19399.365,E2 19399.365} C_VEL
LIN {X 0,Y 267.515,Z 928.626,A -85,B 0,C 180,E1 19406.451,E2 19406.451} C_VEL
LIN {X 0,Y 288.931,Z 895.703,A -85,B 0,C 180,E1 19411.856,E2 19411.856} C_VEL
LIN {X 0,Y 308.542,Z 859.683,A -85,B 0,C 180,E1 19415.774,E2 19415.774} C_VEL
LIN {X 0,Y 309.875,Z 856.048,A -85,B 0,C 180,E1 19416.224,E2 19416.224} C_VEL
LIN {X 0,Y 307.644,Z 839.547,A -85,B 0,C 180,E1 19422.053,E2 19422.053} C_VEL
LIN {X 0,Y 305.17,Z 827.931,A -85,B 0,C 180,E1 19427.822,E2 19427.822} C_VEL
LIN {X 0,Y 303.197,Z 819.895,A -85,B 0,C 180,E1 19434.262,E2 19434.262} C_VEL
LIN {X 0,Y 302.367,Z 817.399,A -85,B 0,C 180,E1 19439.993,E2 19439.993} C_VEL
LIN {X 0,Y 302.524,Z 820.461,A -85,B 0,C 180,E1 19447.18,E2 19447.18} C_VEL
LIN {X 0,Y 303.651,Z 828.328,A -85,B 0,C 180,E1 19453.271,E2 19453.271} C_VEL
LIN {X 0,Y 302.919,Z 834.446,A -85,B 0,C 180,E1 19455.463,E2 19455.463} C_VEL
LIN {X 0,Y 300.631,Z 846.633,A -85,B 0,C 180,E1 19458.962,E2 19458.962} C_VEL
LIN {X 0,Y 300.935,Z 861.081,A -85,B 0,C 180,E1 19464.364,E2 19464.364} C_VEL
LIN {X 0,Y 280.33,Z 895.841,A -85,B 0,C 180,E1 19468.798,E2 19468.798} C_VEL
LIN {X 0,Y 259.502,Z 925.04,A -85,B 0,C 180,E1 19474.311,E2 19474.311} C_VEL
LIN {X 0,Y 239.239,Z 950.079,A -85,B 0,C 180,E1 19481.458,E2 19481.458} C_VEL
LIN {X 0,Y 222.596,Z 969.226,A -85,B 0,C 180,E1 19489.745,E2 19489.745} C_VEL
LIN {X 0,Y 208.784,Z 985.498,A -85,B 0,C 180,E1 19500.977,E2 19500.977} C_VEL
LIN {X 0,Y 201.75,Z 995.319,A -85,B 0,C 180,E1 19512.53,E2 19512.53} C_VEL
LIN {X 0,Y 199.59,Z 999.268,A -85,B 0,C 180,E1 19521.273,E2 19521.273} C_VEL
LIN {X 0,Y 199.456,Z 1000.541,A -85,B 0,C 180,E1 19529.999,E2 19529.999} C_VEL
LIN {X 0,Y 199.715,Z 998.81,A -85,B 0,C 180,E1 19539.857,E2 19539.857} C_VEL
LIN {X 0,Y 203.814,Z 992.205,A -85,B 0,C 180,E1 19551.803,E2 19551.803} C_VEL
LIN {X 0,Y 213.271,Z 980.027,A -85,B 0,C 180,E1 19563.38,E2 19563.38} C_VEL
LIN {X 0,Y 229.981,Z 960.922,A -85,B 0,C 180,E1 19574.164,E2 19574.164} C_VEL
LIN {X 0,Y 250.274,Z 936.696,A -85,B 0,C 180,E1 19582.65,E2 19582.65} C_VEL
LIN {X 0,Y 271.598,Z 908.502,A -85,B 0,C 180,E1 19588.993,E2 19588.993} C_VEL
LIN {X 0,Y 293.56,Z 874.469,A -85,B 0,C 180,E1 19593.963,E2 19593.963} C_VEL
LIN {X 0,Y 300.821,Z 860.805,A -85,B 0,C 180,E1 19595.61,E2 19595.61} C_VEL
LIN {X 0,Y 300.421,Z 844.889,A -85,B 0,C 180,E1 19601.649,E2 19601.649} C_VEL
LIN {X 0,Y 299.258,Z 832.588,A -85,B 0,C 180,E1 19608.333,E2 19608.333} C_VEL
LIN {X 0,Y 298.724,Z 826.162,A -85,B 0,C 180,E1 19614.19,E2 19614.19} C_VEL
LIN {X 0,Y 298.777,Z 824.129,A -85,B 0,C 180,E1 19620.007,E2 19620.007} C_VEL
LIN {X 0,Y 299.793,Z 828.367,A -85,B 0,C 180,E1 19627.26,E2 19627.26} C_VEL
LIN {X 0,Y 301.758,Z 837.684,A -85,B 0,C 180,E1 19633.793,E2 19633.793} C_VEL
LIN {X 0,Y 303.715,Z 850.458,A -85,B 0,C 180,E1 19639.489,E2 19639.489} C_VEL
LIN {X 0,Y 304.629,Z 859.64,A -85,B 0,C 180,E1 19642.703,E2 19642.703} C_VEL
LIN {X 0,Y 300.807,Z 867.731,A -85,B 0,C 180,E1 19643.621,E2 19643.621} C_VEL
LIN {X 0,Y 280.992,Z 901.766,A -85,B 0,C 180,E1 19647.592,E2 19647.592} C_VEL
LIN {X 0,Y 260.797,Z 931.208,A -85,B 0,C 180,E1 19652.669,E2 19652.669} C_VEL
LIN {X 0,Y 239.397,Z 958.832,A -85,B 0,C 180,E1 19659.887,E2 19659.887} C_VEL
LIN {X 0,Y 220.736,Z 981.745,A -85,B 0,C 180,E1 19669.318,E2 19669.318} C_VEL
LIN {X 0,Y 207.346,Z 998.933,A -85,B 0,C 180,E1 19680.638,E2 19680.638} C_VEL
LIN {X 0,Y 200.953,Z 1009.676,A -85,B 0,C 180,E1 19692.46,E2 19692.46} C_VEL
LIN {X 0,Y 199.33,Z 1014.032,A -85,B 0,C 180,E1 19701.263,E2 19701.263} C_VEL
LIN {X 0,Y 199.49,Z 1015.502,A -85,B 0,C 180,E1 19710.001,E2 19710.001} C_VEL
LIN {X 0,Y 199.328,Z 1013.917,A -85,B 0,C 180,E1 19719.062,E2 19719.062} C_VEL
LIN {X 0,Y 201.512,Z 1008.497,A -85,B 0,C 180,E1 19729.163,E2 19729.163} C_VEL
LIN {X 0,Y 208.413,Z 997.531,A -85,B 0,C 180,E1 19740.567,E2 19740.567} C_VEL
LIN {X 0,Y 222.501,Z 979.597,A -85,B 0,C 180,E1 19751.81,E2 19751.81} C_VEL
LIN {X 0,Y 241.397,Z 956.509,A -85,B 0,C 180,E1 19760.876,E2 19760.876} C_VEL
LIN {X 0,Y 263.319,Z 927.966,A -85,B 0,C 180,E1 19768.009,E2 19768.009} C_VEL
LIN {X 0,Y 285.164,Z 895.4,A -85,B 0,C 180,E1 19773.305,E2 19773.305} C_VEL
LIN {X 0,Y 304.188,Z 861.546,A -85,B 0,C 180,E1 19776.963,E2 19776.963} C_VEL
LIN {X 0,Y 304.39,Z 855.99,A -85,B 0,C 180,E1 19778.547,E2 19778.547} C_VEL
LIN {X 0,Y 302.553,Z 841.691,A -85,B 0,C 180,E1 19784.271,E2 19784.271} C_VEL
LIN {X 0,Y 300.666,Z 832.104,A -85,B 0,C 180,E1 19789.843,E2 19789.843} C_VEL
LIN {X 0,Y 299.615,Z 827.132,A -85,B 0,C 180,E1 19794.193,E2 19794.193} C_VEL
LIN {X 0,Y 298.849,Z 824.469,A -85,B 0,C 180,E1 19799.993,E2 19799.993} C_VEL
LIN {X 0,Y 298.894,Z 826.349,A -85,B 0,C 180,E1 19805.807,E2 19805.807} C_VEL
LIN {X 0,Y 299.583,Z 834.995,A -85,B 0,C 180,E1 19813.016,E2 19813.016} C_VEL
LIN {X 0,Y 300.631,Z 846.633,A -85,B 0,C 180,E1 19818.962,E2 19818.962} C_VEL
LIN {X 0,Y 299.401,Z 851.968,A -85,B 0,C 180,E1 19820.276,E2 19820.276} C_VEL
LIN {X 0,Y 295.973,Z 861.988,A -85,B 0,C 180,E1 19822.312,E2 19822.312} C_VEL
LIN {X 0,Y 295.791,Z 865.125,A -85,B 0,C 180,E1 19823.42,E2 19823.42} C_VEL
LIN {X 0,Y 275.455,Z 897.793,A -85,B 0,C 180,E1 19827.582,E2 19827.582} C_VEL
LIN {X 0,Y 252.301,Z 928.851,A -85,B 0,C 180,E1 19833.627,E2 19833.627} C_VEL
LIN {X 0,Y 231.294,Z 953.351,A -85,B 0,C 180,E1 19841.011,E2 19841.011} C_VEL
LIN {X 0,Y 213.342,Z 972.914,A -85,B 0,C 180,E1 19850.302,E2 19850.302} C_VEL
LIN {X 0,Y 200.682,Z 987,A -85,B 0,C 180,E1 19861.03,E2 19861.03} C_VEL
LIN {X 0,Y 194.093,Z 995.62,A -85,B 0,C 180,E1 19871.817,E2 19871.817} C_VEL
LIN {X 0,Y 191.735,Z 999.565,A -85,B 0,C 180,E1 19880.912,E2 19880.912} C_VEL
LIN {X 0,Y 191.569,Z 1000.837,A -85,B 0,C 180,E1 19889.999,E2 19889.999} C_VEL
LIN {X 0,Y 191.715,Z 999.531,A -85,B 0,C 180,E1 19899.087,E2 19899.087} C_VEL
LIN {X 0,Y 194.971,Z 994.248,A -85,B 0,C 180,E1 19910.13,E2 19910.13} C_VEL
LIN {X 0,Y 203.078,Z 984.221,A -85,B 0,C 180,E1 19921.459,E2 19921.459} C_VEL
LIN {X 0,Y 218.179,Z 967.601,A -85,B 0,C 180,E1 19932.579,E2 19932.579} C_VEL
LIN {X 0,Y 238.565,Z 945.026,A -85,B 0,C 180,E1 19941.756,E2 19941.756} C_VEL
LIN {X 0,Y 260.983,Z 917.618,A -85,B 0,C 180,E1 19948.756,E2 19948.756} C_VEL
LIN {X 0,Y 283.22,Z 885.907,A -85,B 0,C 180,E1 19953.998,E2 19953.998} C_VEL
LIN {X 0,Y 295.691,Z 864.757,A -85,B 0,C 180,E1 19956.596,E2 19956.596} C_VEL
LIN {X 0,Y 295.788,Z 849.696,A -85,B 0,C 180,E1 19962.65,E2 19962.65} C_VEL
LIN {X 0,Y 295.194,Z 838.825,A -85,B 0,C 180,E1 19968.919,E2 19968.919} C_VEL
LIN {X 0,Y 294.921,Z 833.221,A -85,B 0,C 180,E1 19974.115,E2 19974.115} C_VEL
LIN {X 0,Y 295.165,Z 831.14,A -85,B 0,C 180,E1 19980.007,E2 19980.007} C_VEL
LIN {X 0,Y 295.787,Z 833.981,A -85,B 0,C 180,E1 19985.882,E2 19985.882} C_VEL
LIN {X 0,Y 297.3,Z 842.451,A -85,B 0,C 180,E1 19992.506,E2 19992.506} C_VEL
LIN {X 0,Y 298.932,Z 855.853,A -85,B 0,C 180,E1 19998.862,E2 19998.862} C_VEL
LIN {X 0,Y 299.434,Z 863.809,A -85,B 0,C 180,E1 20001.795,E2 20001.795} C_VEL
LIN {X 0,Y 278.939,Z 898.958,A -85,B 0,C 180,E1 20005.742,E2 20005.742} C_VEL
LIN {X 0,Y 256.433,Z 930.896,A -85,B 0,C 180,E1 20011.116,E2 20011.116} C_VEL
LIN {X 0,Y 234.187,Z 958.52,A -85,B 0,C 180,E1 20018.337,E2 20018.337} C_VEL
LIN {X 0,Y 214.539,Z 981.434,A -85,B 0,C 180,E1 20027.88,E2 20027.88} C_VEL
LIN {X 0,Y 200.352,Z 998.471,A -85,B 0,C 180,E1 20039.344,E2 20039.344} C_VEL
LIN {X 0,Y 193.252,Z 1009.372,A -85,B 0,C 180,E1 20051.737,E2 20051.737} C_VEL
LIN {X 0,Y 191.452,Z 1013.733,A -85,B 0,C 180,E1 20060.9,E2 20060.9} C_VEL
LIN {X 0,Y 191.601,Z 1015.206,A -85,B 0,C 180,E1 20070.001,E2 20070.001} C_VEL
LIN {X 0,Y 191.453,Z 1013.742,A -85,B 0,C 180,E1 20079.101,E2 20079.101} C_VEL
LIN {X 0,Y 194.131,Z 1007.719,A -85,B 0,C 180,E1 20090.614,E2 20090.614} C_VEL
LIN {X 0,Y 202.446,Z 995.845,A -85,B 0,C 180,E1 20102.836,E2 20102.836} C_VEL
LIN {X 0,Y 216.601,Z 979.021,A -85,B 0,C 180,E1 20113.405,E2 20113.405} C_VEL
LIN {X 0,Y 236.129,Z 956.396,A -85,B 0,C 180,E1 20122.367,E2 20122.367} C_VEL
LIN {X 0,Y 259.063,Z 927.66,A -85,B 0,C 180,E1 20129.55,E2 20129.55} C_VEL
LIN {X 0,Y 281.32,Z 895.584,A -85,B 0,C 180,E1 20134.718,E2 20134.718} C_VEL
LIN {X 0,Y 299.533,Z 863.909,A -85,B 0,C 180,E1 20138.207,E2 20138.207} C_VEL
LIN {X 0,Y 298.355,Z 849.395,A -85,B 0,C 180,E1 20143.939,E2 20143.939} C_VEL
LIN {X 0,Y 296.765,Z 839.413,A -85,B 0,C 180,E1 20149.616,E2 20149.616} C_VEL
LIN {X 0,Y 295.844,Z 834.27,A -85,B 0,C 180,E1 20154.119,E2 20154.119} C_VEL
LIN {X 0,Y 295.22,Z 831.475,A -85,B 0,C 180,E1 20159.993,E2 20159.993} C_VEL
LIN {X 0,Y 295.066,Z 833.437,A -85,B 0,C 180,E1 20165.882,E2 20165.882} C_VEL
LIN {X 0,Y 295.481,Z 842.292,A -85,B 0,C 180,E1 20173.196,E2 20173.196} C_VEL
LIN {X 0,Y 296.016,Z 854.597,A -85,B 0,C 180,E1 20179.408,E2 20179.408} C_VEL
LIN {X 0,Y 295.973,Z 861.988,A -85,B 0,C 180,E1 20182.312,E2 20182.312} C_VEL
LIN {X 0,Y 293.604,Z 867.033,A -85,B 0,C 180,E1 20183.082,E2 20183.082} C_VEL
LIN {X 0,Y 283.35,Z 880.762,A -85,B 0,C 180,E1 20183.71,E2 20183.71} C_VEL
LIN {X 0,Y 261.721,Z 911.762,A -85,B 0,C 180,E1 20188.391,E2 20188.391} C_VEL
LIN {X 0,Y 238.992,Z 939.389,A -85,B 0,C 180,E1 20194.746,E2 20194.746} C_VEL
LIN {X 0,Y 217.727,Z 962.38,A -85,B 0,C 180,E1 20203.098,E2 20203.098} C_VEL
LIN {X 0,Y 199.783,Z 980.774,A -85,B 0,C 180,E1 20214.03,E2 20214.03} C_VEL
LIN {X 0,Y 188.867,Z 992.907,A -85,B 0,C 180,E1 20226.369,E2 20226.369} C_VEL
LIN {X 0,Y 184.908,Z 998.23,A -85,B 0,C 180,E1 20235.779,E2 20235.779} C_VEL
LIN {X 0,Y 183.511,Z 1000.828,A -85,B 0,C 180,E1 20245.266,E2 20245.266} C_VEL
LIN {X 0,Y 183.665,Z 1001.133,A -85,B 0,C 180,E1 20249.999,E2 20249.999} C_VEL
LIN {X 0,Y 183.865,Z 999.829,A -85,B 0,C 180,E1 20259.479,E2 20259.479} C_VEL
LIN {X 0,Y 187.324,Z 994.68,A -85,B 0,C 180,E1 20270.777,E2 20270.777} C_VEL
LIN {X 0,Y 196.167,Z 984.528,A -85,B 0,C 180,E1 20282.702,E2 20282.702} C_VEL
LIN {X 0,Y 212.276,Z 967.907,A -85,B 0,C 180,E1 20294.06,E2 20294.06} C_VEL
LIN {X 0,Y 233.593,Z 945.335,A -85,B 0,C 180,E1 20303.331,E2 20303.331} C_VEL
LIN {X 0,Y 256.865,Z 917.922,A -85,B 0,C 180,E1 20310.307,E2 20310.307} C_VEL
LIN {X 0,Y 279.803,Z 886.211,A -85,B 0,C 180,E1 20315.472,E2 20315.472} C_VEL
LIN {X 0,Y 290.534,Z 868.661,A -85,B 0,C 180,E1 20317.611,E2 20317.611} C_VEL
LIN {X 0,Y 291.122,Z 855.024,A -85,B 0,C 180,E1 20323.388,E2 20323.388} C_VEL
LIN {X 0,Y 290.947,Z 844.944,A -85,B 0,C 180,E1 20329.514,E2 20329.514} C_VEL
LIN {X 0,Y 291.031,Z 840.26,A -85,B 0,C 180,E1 20334.036,E2 20334.036} C_VEL
LIN {X 0,Y 291.324,Z 838.055,A -85,B 0,C 180,E1 20340.007,E2 20340.007} C_VEL
LIN {X 0,Y 291.879,Z 841.053,A -85,B 0,C 180,E1 20345.961,E2 20345.961} C_VEL
LIN {X 0,Y 293.071,Z 849.7,A -85,B 0,C 180,E1 20352.689,E2 20352.689} C_VEL
LIN {X 0,Y 294.129,Z 862.438,A -85,B 0,C 180,E1 20358.743,E2 20358.743} C_VEL
LIN {X 0,Y 293.752,Z 868.866,A -85,B 0,C 180,E1 20360.901,E2 20360.901} C_VEL
LIN {X 0,Y 273.013,Z 902.32,A -85,B 0,C 180,E1 20364.722,E2 20364.722} C_VEL
LIN {X 0,Y 250.983,Z 932.211,A -85,B 0,C 180,E1 20369.868,E2 20369.868} C_VEL
LIN {X 0,Y 229.759,Z 957.557,A -85,B 0,C 180,E1 20376.499,E2 20376.499} C_VEL
LIN {X 0,Y 209.561,Z 979.97,A -85,B 0,C 180,E1 20385.716,E2 20385.716} C_VEL
LIN {X 0,Y 193.488,Z 997.977,A -85,B 0,C 180,E1 20397.927,E2 20397.927} C_VEL
LIN {X 0,Y 185.575,Z 1009.068,A -85,B 0,C 180,E1 20410.953,E2 20410.953} C_VEL
LIN {X 0,Y 183.421,Z 1013.821,A -85,B 0,C 180,E1 20422.147,E2 20422.147} C_VEL
LIN {X 0,Y 183.693,Z 1014.91,A -85,B 0,C 180,E1 20430.001,E2 20430.001} C_VEL
LIN {X 0,Y 183.584,Z 1013.443,A -85,B 0,C 180,E1 20439.495,E2 20439.495} C_VEL
LIN {X 0,Y 186.526,Z 1007.414,A -85,B 0,C 180,E1 20451.495,E2 20451.495} C_VEL
LIN {X 0,Y 195.511,Z 995.621,A -85,B 0,C 180,E1 20464.076,E2 20464.076} C_VEL
LIN {X 0,Y 210.645,Z 978.718,A -85,B 0,C 180,E1 20474.952,E2 20474.952} C_VEL
LIN {X 0,Y 231.552,Z 955.674,A -85,B 0,C 180,E1 20484.106,E2 20484.106} C_VEL
LIN {X 0,Y 254.973,Z 927.353,A -85,B 0,C 180,E1 20491.151,E2 20491.151} C_VEL
LIN {X 0,Y 278.155,Z 894.945,A -85,B 0,C 180,E1 20496.276,E2 20496.276} C_VEL
LIN {X 0,Y 294.386,Z 867.492,A -85,B 0,C 180,E1 20499.365,E2 20499.365} C_VEL
LIN {X 0,Y 293.638,Z 854.022,A -85,B 0,C 180,E1 20505.054,E2 20505.054} C_VEL
LIN {X 0,Y 292.394,Z 844.57,A -85,B 0,C 180,E1 20511.057,E2 20511.057} C_VEL
LIN {X 0,Y 291.56,Z 839.335,A -85,B 0,C 180,E1 20517.016,E2 20517.016} C_VEL
LIN {X 0,Y 291.385,Z 838.382,A -85,B 0,C 180,E1 20519.993,E2 20519.993} C_VEL
LIN {X 0,Y 291.168,Z 840.495,A -85,B 0,C 180,E1 20525.962,E2 20525.962} C_VEL
LIN {X 0,Y 291.115,Z 848.398,A -85,B 0,C 180,E1 20532.697,E2 20532.697} C_VEL
LIN {X 0,Y 291.144,Z 860.6,A -85,B 0,C 180,E1 20539.053,E2 20539.053} C_VEL
LIN {X 0,Y 290.405,Z 869.351,A -85,B 0,C 180,E1 20542.424,E2 20542.424} C_VEL
LIN {X 0,Y 283.35,Z 880.762,A -85,B 0,C 180,E1 20543.71,E2 20543.71} C_VEL
LIN {X 0,Y 272.9,Z 894.101,A -85,B 0,C 180,E1 20544.702,E2 20544.702} C_VEL
LIN {X 0,Y 262.132,Z 906.695,A -85,B 0,C 180,E1 20545.865,E2 20545.865} C_VEL
LIN {X 0,Y 238.562,Z 935.19,A -85,B 0,C 180,E1 20551.909,E2 20551.909} C_VEL
LIN {X 0,Y 216.317,Z 958.51,A -85,B 0,C 180,E1 20559.651,E2 20559.651} C_VEL
LIN {X 0,Y 198.298,Z 976.199,A -85,B 0,C 180,E1 20569.064,E2 20569.064} C_VEL
LIN {X 0,Y 184.887,Z 989.469,A -85,B 0,C 180,E1 20580.569,E2 20580.569} C_VEL
LIN {X 0,Y 177.93,Z 997.383,A -85,B 0,C 180,E1 20592.672,E2 20592.672} C_VEL
LIN {X 0,Y 175.632,Z 1001.124,A -85,B 0,C 180,E1 20605.054,E2 20605.054} C_VEL
LIN {X 0,Y 175.761,Z 1001.429,A -85,B 0,C 180,E1 20609.999,E2 20609.999} C_VEL
LIN {X 0,Y 176.014,Z 1000.128,A -85,B 0,C 180,E1 20619.906,E2 20619.906} C_VEL
LIN {X 0,Y 180.245,Z 994.466,A -85,B 0,C 180,E1 20632.53,E2 20632.53} C_VEL
LIN {X 0,Y 190.621,Z 983.539,A -85,B 0,C 180,E1 20645.159,E2 20645.159} C_VEL
LIN {X 0,Y 207.867,Z 966.884,A -85,B 0,C 180,E1 20656.292,E2 20656.292} C_VEL
LIN {X 0,Y 229.663,Z 944.727,A -85,B 0,C 180,E1 20665.247,E2 20665.247} C_VEL
LIN {X 0,Y 252.835,Z 918.371,A -85,B 0,C 180,E1 20671.875,E2 20671.875} C_VEL
LIN {X 0,Y 276.551,Z 886.518,A -85,B 0,C 180,E1 20676.992,E2 20676.992} C_VEL
LIN {X 0,Y 285.48,Z 872.17,A -85,B 0,C 180,E1 20678.834,E2 20678.834} C_VEL
LIN {X 0,Y 286.406,Z 859.338,A -85,B 0,C 180,E1 20684.683,E2 20684.683} C_VEL
LIN {X 0,Y 286.654,Z 850.179,A -85,B 0,C 180,E1 20690.891,E2 20690.891} C_VEL
LIN {X 0,Y 286.851,Z 847.166,A -85,B 0,C 180,E1 20693.948,E2 20693.948} C_VEL
LIN {X 0,Y 287.357,Z 844.906,A -85,B 0,C 180,E1 20700.007,E2 20700.007} C_VEL
LIN {X 0,Y 287.766,Z 847.995,A -85,B 0,C 180,E1 20706.047,E2 20706.047} C_VEL
LIN {X 0,Y 288.603,Z 855.629,A -85,B 0,C 180,E1 20712.119,E2 20712.119} C_VEL
LIN {X 0,Y 289.167,Z 868.197,A -85,B 0,C 180,E1 20718.315,E2 20718.315} C_VEL
LIN {X 0,Y 288.695,Z 872.514,A -85,B 0,C 180,E1 20719.771,E2 20719.771} C_VEL
LIN {X 0,Y 266.366,Z 906.86,A -85,B 0,C 180,E1 20723.825,E2 20723.825} C_VEL
LIN {X 0,Y 241.621,Z 938.456,A -85,B 0,C 180,E1 20729.651,E2 20729.651} C_VEL
LIN {X 0,Y 217.423,Z 965.276,A -85,B 0,C 180,E1 20737.617,E2 20737.617} C_VEL
LIN {X 0,Y 197.404,Z 986.17,A -85,B 0,C 180,E1 20747.847,E2 20747.847} C_VEL
LIN {X 0,Y 183.356,Z 1001.408,A -85,B 0,C 180,E1 20760.301,E2 20760.301} C_VEL
LIN {X 0,Y 177.11,Z 1010.052,A -85,B 0,C 180,E1 20772.591,E2 20772.591} C_VEL
LIN {X 0,Y 175.501,Z 1014.232,A -85,B 0,C 180,E1 20785.052,E2 20785.052} C_VEL
LIN {X 0,Y 175.784,Z 1014.613,A -85,B 0,C 180,E1 20790.001,E2 20790.001} C_VEL
LIN {X 0,Y 175.697,Z 1013.143,A -85,B 0,C 180,E1 20799.926,E2 20799.926} C_VEL
LIN {X 0,Y 179.098,Z 1006.945,A -85,B 0,C 180,E1 20812.698,E2 20812.698} C_VEL
LIN {X 0,Y 187.588,Z 996.609,A -85,B 0,C 180,E1 20824.403,E2 20824.403} C_VEL
LIN {X 0,Y 203.837,Z 979.513,A -85,B 0,C 180,E1 20836.038,E2 20836.038} C_VEL
LIN {X 0,Y 225.827,Z 956.482,A -85,B 0,C 180,E1 20845.453,E2 20845.453} C_VEL
LIN {X 0,Y 251.099,Z 927.047,A -85,B 0,C 180,E1 20852.799,E2 20852.799} C_VEL
LIN {X 0,Y 275.056,Z 894.529,A -85,B 0,C 180,E1 20857.842,E2 20857.842} C_VEL
LIN {X 0,Y 289.296,Z 871.568,A -85,B 0,C 180,E1 20860.403,E2 20860.403} C_VEL
LIN {X 0,Y 288.934,Z 858.419,A -85,B 0,C 180,E1 20866.355,E2 20866.355} C_VEL
LIN {X 0,Y 287.941,Z 849.813,A -85,B 0,C 180,E1 20872.44,E2 20872.44} C_VEL
LIN {X 0,Y 287.542,Z 846.211,A -85,B 0,C 180,E1 20876.975,E2 20876.975} C_VEL
LIN {X 0,Y 287.406,Z 845.223,A -85,B 0,C 180,E1 20879.993,E2 20879.993} C_VEL
LIN {X 0,Y 286.971,Z 847.406,A -85,B 0,C 180,E1 20886.049,E2 20886.049} C_VEL
LIN {X 0,Y 286.658,Z 855.622,A -85,B 0,C 180,E1 20892.963,E2 20892.963} C_VEL
LIN {X 0,Y 286.223,Z 866.092,A -85,B 0,C 180,E1 20898.495,E2 20898.495} C_VEL
LIN {X 0,Y 285.133,Z 873.467,A -85,B 0,C 180,E1 20901.355,E2 20901.355} C_VEL
LIN {X 0,Y 262.737,Z 905.888,A -85,B 0,C 180,E1 20905.734,E2 20905.734} C_VEL
LIN {X 0,Y 262.132,Z 906.695,A -85,B 0,C 180,E1 20905.865,E2 20905.865} C_VEL
LIN {X 0,Y 250.945,Z 918.82,A -85,B 0,C 180,E1 20907.217,E2 20907.217} C_VEL
LIN {X 0,Y 239.411,Z 930.023,A -85,B 0,C 180,E1 20908.832,E2 20908.832} C_VEL
LIN {X 0,Y 214.732,Z 955.562,A -85,B 0,C 180,E1 20916.622,E2 20916.622} C_VEL
LIN {X 0,Y 193.335,Z 975.498,A -85,B 0,C 180,E1 20926.744,E2 20926.744} C_VEL
LIN {X 0,Y 177.868,Z 989.772,A -85,B 0,C 180,E1 20939.285,E2 20939.285} C_VEL
LIN {X 0,Y 170.273,Z 997.684,A -85,B 0,C 180,E1 20951.866,E2 20951.866} C_VEL
LIN {X 0,Y 167.729,Z 1001.422,A -85,B 0,C 180,E1 20964.82,E2 20964.82} C_VEL
LIN {X 0,Y 167.856,Z 1001.726,A -85,B 0,C 180,E1 20969.999,E2 20969.999} C_VEL
LIN {X 0,Y 168.201,Z 1000.426,A -85,B 0,C 180,E1 20980.371,E2 20980.371} C_VEL
LIN {X 0,Y 172.811,Z 994.769,A -85,B 0,C 180,E1 20993.556,E2 20993.556} C_VEL
LIN {X 0,Y 184.014,Z 983.845,A -85,B 0,C 180,E1 21006.621,E2 21006.621} C_VEL
LIN {X 0,Y 201.103,Z 968.354,A -85,B 0,C 180,E1 21017.365,E2 21017.365} C_VEL
LIN {X 0,Y 224.473,Z 945.717,A -85,B 0,C 180,E1 21026.741,E2 21026.741} C_VEL
LIN {X 0,Y 249.528,Z 918.158,A -85,B 0,C 180,E1 21033.624,E2 21033.624} C_VEL
LIN {X 0,Y 273.515,Z 886.823,A -85,B 0,C 180,E1 21038.54,E2 21038.54} C_VEL
LIN {X 0,Y 279.966,Z 877.198,A -85,B 0,C 180,E1 21039.685,E2 21039.685} C_VEL
LIN {X 0,Y 281.587,Z 866.519,A -85,B 0,C 180,E1 21044.414,E2 21044.414} C_VEL
LIN {X 0,Y 282.241,Z 857.022,A -85,B 0,C 180,E1 21050.785,E2 21050.785} C_VEL
LIN {X 0,Y 282.628,Z 854.041,A -85,B 0,C 180,E1 21053.858,E2 21053.858} C_VEL
LIN {X 0,Y 283.213,Z 851.629,A -85,B 0,C 180,E1 21060.007,E2 21060.007} C_VEL
LIN {X 0,Y 283.547,Z 854.877,A -85,B 0,C 180,E1 21066.137,E2 21066.137} C_VEL
LIN {X 0,Y 284.007,Z 862.709,A -85,B 0,C 180,E1 21072.318,E2 21072.318} C_VEL
LIN {X 0,Y 284.041,Z 874.765,A -85,B 0,C 180,E1 21078.255,E2 21078.255} C_VEL
LIN {X 0,Y 281.232,Z 879.955,A -85,B 0,C 180,E1 21078.987,E2 21078.987} C_VEL
LIN {X 0,Y 259.037,Z 911.899,A -85,B 0,C 180,E1 21082.988,E2 21082.988} C_VEL
LIN {X 0,Y 235.243,Z 940.791,A -85,B 0,C 180,E1 21088.565,E2 21088.565} C_VEL
LIN {X 0,Y 211.324,Z 966.074,A -85,B 0,C 180,E1 21096.291,E2 21096.291} C_VEL
LIN {X 0,Y 191.372,Z 985.859,A -85,B 0,C 180,E1 21106.191,E2 21106.191} C_VEL
LIN {X 0,Y 175.954,Z 1001.471,A -85,B 0,C 180,E1 21119.383,E2 21119.383} C_VEL
LIN {X 0,Y 169.429,Z 1009.748,A -85,B 0,C 180,E1 21131.775,E2 21131.775} C_VEL
LIN {X 0,Y 167.582,Z 1013.934,A -85,B 0,C 180,E1 21144.817,E2 21144.817} C_VEL
LIN {X 0,Y 167.874,Z 1014.316,A -85,B 0,C 180,E1 21150.001,E2 21150.001} C_VEL
LIN {X 0,Y 167.829,Z 1012.844,A -85,B 0,C 180,E1 21160.396,E2 21160.396} C_VEL
LIN {X 0,Y 171.447,Z 1006.851,A -85,B 0,C 180,E1 21173.417,E2 21173.417} C_VEL
LIN {X 0,Y 180.846,Z 996.301,A -85,B 0,C 180,E1 21185.879,E2 21185.879} C_VEL
LIN {X 0,Y 198.722,Z 978.662,A -85,B 0,C 180,E1 21198.035,E2 21198.035} C_VEL
LIN {X 0,Y 221.662,Z 955.737,A -85,B 0,C 180,E1 21207.349,E2 21207.349} C_VEL
LIN {X 0,Y 247.669,Z 926.465,A -85,B 0,C 180,E1 21214.544,E2 21214.544} C_VEL
LIN {X 0,Y 272.358,Z 893.806,A -85,B 0,C 180,E1 21219.485,E2 21219.485} C_VEL
LIN {X 0,Y 284.142,Z 875.179,A -85,B 0,C 180,E1 21221.611,E2 21221.611} C_VEL
LIN {X 0,Y 284.126,Z 862.825,A -85,B 0,C 180,E1 21227.687,E2 21227.687} C_VEL
LIN {X 0,Y 283.591,Z 855.168,A -85,B 0,C 180,E1 21233.864,E2 21233.864} C_VEL
LIN {X 0,Y 283.263,Z 851.948,A -85,B 0,C 180,E1 21239.993,E2 21239.993} C_VEL
LIN {X 0,Y 282.728,Z 854.3,A -85,B 0,C 180,E1 21246.14,E2 21246.14} C_VEL
LIN {X 0,Y 281.992,Z 862.778,A -85,B 0,C 180,E1 21253.26,E2 21253.26} C_VEL
LIN {X 0,Y 280.939,Z 873.54,A -85,B 0,C 180,E1 21258.856,E2 21258.856} C_VEL
LIN {X 0,Y 279.975,Z 877.433,A -85,B 0,C 180,E1 21260.238,E2 21260.238} C_VEL
LIN {X 0,Y 255.703,Z 910.822,A -85,B 0,C 180,E1 21264.902,E2 21264.902} C_VEL
LIN {X 0,Y 239.411,Z 930.023,A -85,B 0,C 180,E1 21268.832,E2 21268.832} C_VEL
LIN {X 0,Y 227.591,Z 940.603,A -85,B 0,C 180,E1 21270.694,E2 21270.694} C_VEL
LIN {X 0,Y 215.716,Z 950.375,A -85,B 0,C 180,E1 21272.831,E2 21272.831} C_VEL
LIN {X 0,Y 193.07,Z 970.908,A -85,B 0,C 180,E1 21281.998,E2 21281.998} C_VEL
LIN {X 0,Y 174.329,Z 987.008,A -85,B 0,C 180,E1 21294.459,E2 21294.459} C_VEL
LIN {X 0,Y 163.817,Z 996.825,A -85,B 0,C 180,E1 21308.302,E2 21308.302} C_VEL
LIN {X 0,Y 160.371,Z 1000.758,A -85,B 0,C 180,E1 21319.115,E2 21319.115} C_VEL
LIN {X 0,Y 159.97,Z 1002.022,A -85,B 0,C 180,E1 21329.999,E2 21329.999} C_VEL
LIN {X 0,Y 160.365,Z 1000.725,A -85,B 0,C 180,E1 21340.883,E2 21340.883} C_VEL
LIN {X 0,Y 165.532,Z 994.993,A -85,B 0,C 180,E1 21354.812,E2 21354.812} C_VEL
LIN {X 0,Y 177.558,Z 984.151,A -85,B 0,C 180,E1 21368.186,E2 21368.186} C_VEL
LIN {X 0,Y 195.678,Z 968.661,A -85,B 0,C 180,E1 21379.12,E2 21379.12} C_VEL
LIN {X 0,Y 219.66,Z 946.495,A -85,B 0,C 180,E1 21388.365,E2 21388.365} C_VEL
LIN {X 0,Y 246.05,Z 918.442,A -85,B 0,C 180,E1 21395.322,E2 21395.322} C_VEL
LIN {X 0,Y 270.932,Z 886.725,A -85,B 0,C 180,E1 21400.184,E2 21400.184} C_VEL
LIN {X 0,Y 275.345,Z 880.148,A -85,B 0,C 180,E1 21401.013,E2 21401.013} C_VEL
LIN {X 0,Y 276.889,Z 869.977,A -85,B 0,C 180,E1 21406.22,E2 21406.22} C_VEL
LIN {X 0,Y 277.819,Z 862.374,A -85,B 0,C 180,E1 21412.018,E2 21412.018} C_VEL
LIN {X 0,Y 278.412,Z 859.043,A -85,B 0,C 180,E1 21416.891,E2 21416.891} C_VEL
LIN {X 0,Y 278.913,Z 858.281,A -85,B 0,C 180,E1 21420.008,E2 21420.008} C_VEL
LIN {X 0,Y 279.078,Z 861.618,A -85,B 0,C 180,E1 21426.236,E2 21426.236} C_VEL
LIN {X 0,Y 279.299,Z 869.787,A -85,B 0,C 180,E1 21432.529,E2 21432.529} C_VEL
LIN {X 0,Y 278.949,Z 878.854,A -85,B 0,C 180,E1 21437.184,E2 21437.184} C_VEL
LIN {X 0,Y 255.969,Z 911.591,A -85,B 0,C 180,E1 21441.312,E2 21441.312} C_VEL
LIN {X 0,Y 232.119,Z 939.728,A -85,B 0,C 180,E1 21446.591,E2 21446.591} C_VEL
LIN {X 0,Y 206.407,Z 965.887,A -85,B 0,C 180,E1 21454.494,E2 21454.494} C_VEL
LIN {X 0,Y 185.504,Z 985.549,A -85,B 0,C 180,E1 21464.425,E2 21464.425} C_VEL
LIN {X 0,Y 168.645,Z 1001.425,A -85,B 0,C 180,E1 21478.293,E2 21478.293} C_VEL
LIN {X 0,Y 161.692,Z 1009.569,A -85,B 0,C 180,E1 21491.145,E2 21491.145} C_VEL
LIN {X 0,Y 159.687,Z 1013.637,A -85,B 0,C 180,E1 21504.56,E2 21504.56} C_VEL
LIN {X 0,Y 159.985,Z 1014.02,A -85,B 0,C 180,E1 21510.001,E2 21510.001} C_VEL
LIN {X 0,Y 159.955,Z 1012.543,A -85,B 0,C 180,E1 21520.914,E2 21520.914} C_VEL
LIN {X 0,Y 164.003,Z 1006.546,A -85,B 0,C 180,E1 21534.548,E2 21534.548} C_VEL
LIN {X 0,Y 175.415,Z 994.82,A -85,B 0,C 180,E1 21548.501,E2 21548.501} C_VEL
LIN {X 0,Y 193.207,Z 978.424,A -85,B 0,C 180,E1 21559.825,E2 21559.825} C_VEL
LIN {X 0,Y 217.831,Z 954.904,A -85,B 0,C 180,E1 21569.335,E2 21569.335} C_VEL
LIN {X 0,Y 244.261,Z 926.161,A -85,B 0,C 180,E1 21576.279,E2 21576.279} C_VEL
LIN {X 0,Y 269.347,Z 893.891,A -85,B 0,C 180,E1 21581.064,E2 21581.064} C_VEL
LIN {X 0,Y 278.825,Z 879.727,A -85,B 0,C 180,E1 21582.592,E2 21582.592} C_VEL
LIN {X 0,Y 279.431,Z 869.881,A -85,B 0,C 180,E1 21587.477,E2 21587.477} C_VEL
LIN {X 0,Y 279.107,Z 861.904,A -85,B 0,C 180,E1 21593.765,E2 21593.765} C_VEL
LIN {X 0,Y 278.962,Z 858.573,A -85,B 0,C 180,E1 21599.992,E2 21599.992} C_VEL
LIN {X 0,Y 278.193,Z 861.007,A -85,B 0,C 180,E1 21606.241,E2 21606.241} C_VEL
LIN {X 0,Y 277.254,Z 868.375,A -85,B 0,C 180,E1 21612.608,E2 21612.608} C_VEL
LIN {X 0,Y 275.766,Z 878.97,A -85,B 0,C 180,E1 21618.359,E2 21618.359} C_VEL
LIN {X 0,Y 275.088,Z 880.916,A -85,B 0,C 180,E1 21619.036,E2 21619.036} C_VEL
LIN {X 0,Y 251.781,Z 911.851,A -85,B 0,C 180,E1 21623.367,E2 21623.367} C_VEL
LIN {X 0,Y 226.36,Z 939.977,A -85,B 0,C 180,E1 21629.592,E2 21629.592} C_VEL
LIN {X 0,Y 215.716,Z 950.375,A -85,B 0,C 180,E1 21632.831,E2 21632.831} C_VEL
LIN {X 0,Y 203.744,Z 959.447,A -85,B 0,C 180,E1 21635.325,E2 21635.325} C_VEL
LIN {X 0,Y 191.972,Z 967.686,A -85,B 0,C 180,E1 21638.206,E2 21638.206} C_VEL
LIN {X 0,Y 172.461,Z 983.528,A -85,B 0,C 180,E1 21649.127,E2 21649.127} C_VEL
LIN {X 0,Y 159.711,Z 994.118,A -85,B 0,C 180,E1 21661.704,E2 21661.704} C_VEL
LIN {X 0,Y 154.04,Z 999.431,A -85,B 0,C 180,E1 21672.849,E2 21672.849} C_VEL
LIN {X 0,Y 151.926,Z 1002.058,A -85,B 0,C 180,E1 21685.012,E2 21685.012} C_VEL
LIN {X 0,Y 151.874,Z 1002.063,A -85,B 0,C 180,E1 21694.757,E2 21694.757} C_VEL
LIN {X 0,Y 154.044,Z 999.381,A -85,B 0,C 180,E1 21707.148,E2 21707.148} C_VEL
LIN {X 0,Y 161.8,Z 992.179,A -85,B 0,C 180,E1 21720.975,E2 21720.975} C_VEL
LIN {X 0,Y 178.138,Z 978.946,A -85,B 0,C 180,E1 21734.523,E2 21734.523} C_VEL
LIN {X 0,Y 200.483,Z 960.297,A -85,B 0,C 180,E1 21745.214,E2 21745.214} C_VEL
LIN {X 0,Y 225.319,Z 937.281,A -85,B 0,C 180,E1 21752.917,E2 21752.917} C_VEL
LIN {X 0,Y 251.598,Z 908.499,A -85,B 0,C 180,E1 21758.846,E2 21758.846} C_VEL
LIN {X 0,Y 270.354,Z 884.027,A -85,B 0,C 180,E1 21762.186,E2 21762.186} C_VEL
LIN {X 0,Y 272.085,Z 875.061,A -85,B 0,C 180,E1 21767.149,E2 21767.149} C_VEL
LIN {X 0,Y 273.519,Z 867.432,A -85,B 0,C 180,E1 21773.652,E2 21773.652} C_VEL
LIN {X 0,Y 274.468,Z 864.812,A -85,B 0,C 180,E1 21780.008,E2 21780.008} C_VEL
LIN {X 0,Y 274.541,Z 868.324,A -85,B 0,C 180,E1 21786.339,E2 21786.339} C_VEL
LIN {X 0,Y 274.36,Z 875.32,A -85,B 0,C 180,E1 21791.95,E2 21791.95} C_VEL
LIN {X 0,Y 273.917,Z 882.923,A -85,B 0,C 180,E1 21796.05,E2 21796.05} C_VEL
LIN {X 0,Y 248.442,Z 917.087,A -85,B 0,C 180,E1 21800.448,E2 21800.448} C_VEL
LIN {X 0,Y 220.49,Z 947.728,A -85,B 0,C 180,E1 21806.787,E2 21806.787} C_VEL
LIN {X 0,Y 194.237,Z 972.54,A -85,B 0,C 180,E1 21815.536,E2 21815.536} C_VEL
LIN {X 0,Y 172.199,Z 991.712,A -85,B 0,C 180,E1 21827.325,E2 21827.325} C_VEL
LIN {X 0,Y 158.237,Z 1004.545,A -85,B 0,C 180,E1 21841.419,E2 21841.419} C_VEL
LIN {X 0,Y 153.25,Z 1010.405,A -85,B 0,C 180,E1 21852.76,E2 21852.76} C_VEL
LIN {X 0,Y 151.748,Z 1013.481,A -85,B 0,C 180,E1 21866.254,E2 21866.254} C_VEL
LIN {X 0,Y 151.743,Z 1013.485,A -85,B 0,C 180,E1 21873.717,E2 21873.717} C_VEL
LIN {X 0,Y 153.249,Z 1010.423,A -85,B 0,C 180,E1 21887.242,E2 21887.242} C_VEL
LIN {X 0,Y 160.66,Z 1002.095,A -85,B 0,C 180,E1 21901.975,E2 21901.975} C_VEL
LIN {X 0,Y 175.673,Z 988.74,A -85,B 0,C 180,E1 21915.005,E2 21915.005} C_VEL
LIN {X 0,Y 198.256,Z 969.017,A -85,B 0,C 180,E1 21926.023,E2 21926.023} C_VEL
LIN {X 0,Y 223.985,Z 944.298,A -85,B 0,C 180,E1 21934.108,E2 21934.108} C_VEL
LIN {X 0,Y 250.011,Z 915.339,A -85,B 0,C 180,E1 21939.835,E2 21939.835} C_VEL
LIN {X 0,Y 274.051,Z 882.982,A -85,B 0,C 180,E1 21943.958,E2 21943.958} C_VEL
LIN {X 0,Y 274.548,Z 873.065,A -85,B 0,C 180,E1 21949.669,E2 21949.669} C_VEL
LIN {X 0,Y 274.554,Z 867.276,A -85,B 0,C 180,E1 21955.248,E2 21955.248} C_VEL
LIN {X 0,Y 274.506,Z 865.12,A -85,B 0,C 180,E1 21959.992,E2 21959.992} C_VEL
LIN {X 0,Y 273.59,Z 867.699,A -85,B 0,C 180,E1 21966.346,E2 21966.346} C_VEL
LIN {X 0,Y 272.244,Z 875.234,A -85,B 0,C 180,E1 21972.844,E2 21972.844} C_VEL
LIN {X 0,Y 270.32,Z 884.401,A -85,B 0,C 180,E1 21977.788,E2 21977.788} C_VEL
LIN {X 0,Y 246.831,Z 914.27,A -85,B 0,C 180,E1 21982.029,E2 21982.029} C_VEL
LIN {X 0,Y 220.884,Z 941.761,A -85,B 0,C 180,E1 21988.191,E2 21988.191} C_VEL
LIN {X 0,Y 196.814,Z 963.601,A -85,B 0,C 180,E1 21996.121,E2 21996.121} C_VEL
LIN {X 0,Y 191.972,Z 967.686,A -85,B 0,C 180,E1 21998.206,E2 21998.206} C_VEL
LIN {X 0,Y 180.411,Z 975.15,A -85,B 0,C 180,E1 22001.55,E2 22001.55} C_VEL
LIN {X 0,Y 169.231,Z 981.749,A -85,B 0,C 180,E1 22005.417,E2 22005.417} C_VEL
LIN {X 0,Y 152.633,Z 994.421,A -85,B 0,C 180,E1 22020.264,E2 22020.264} C_VEL
LIN {X 0,Y 146.39,Z 999.731,A -85,B 0,C 180,E1 22031.922,E2 22031.922} C_VEL
LIN {X 0,Y 144.049,Z 1002.313,A -85,B 0,C 180,E1 22043.965,E2 22043.965} C_VEL
LIN {X 0,Y 144.178,Z 1002.614,A -85,B 0,C 180,E1 22049.999,E2 22049.999} C_VEL
LIN {X 0,Y 144.752,Z 1001.323,A -85,B 0,C 180,E1 22062.074,E2 22062.074} C_VEL
LIN {X 0,Y 150.677,Z 995.864,A -85,B 0,C 180,E1 22076.883,E2 22076.883} C_VEL
LIN {X 0,Y 163.402,Z 986.06,A -85,B 0,C 180,E1 22090.436,E2 22090.436} C_VEL
LIN {X 0,Y 185.33,Z 969.35,A -85,B 0,C 180,E1 22102.892,E2 22102.892} C_VEL
LIN {X 0,Y 211.672,Z 947.016,A -85,B 0,C 180,E1 22112.15,E2 22112.15} C_VEL
LIN {X 0,Y 239.539,Z 919.286,A -85,B 0,C 180,E1 22118.798,E2 22118.798} C_VEL
LIN {X 0,Y 265.449,Z 887.888,A -85,B 0,C 180,E1 22123.44,E2 22123.44} C_VEL
LIN {X 0,Y 267.705,Z 878.289,A -85,B 0,C 180,E1 22129.418,E2 22129.418} C_VEL
LIN {X 0,Y 268.663,Z 873.959,A -85,B 0,C 180,E1 22133.537,E2 22133.537} C_VEL
LIN {X 0,Y 269.858,Z 871.234,A -85,B 0,C 180,E1 22140.008,E2 22140.008} C_VEL
LIN {X 0,Y 269.761,Z 874.797,A -85,B 0,C 180,E1 22146.452,E2 22146.452} C_VEL
LIN {X 0,Y 269.343,Z 882.149,A -85,B 0,C 180,E1 22152.176,E2 22152.176} C_VEL
LIN {X 0,Y 268.775,Z 886.98,A -85,B 0,C 180,E1 22154.926,E2 22154.926} C_VEL
LIN {X 0,Y 243.905,Z 918.804,A -85,B 0,C 180,E1 22158.988,E2 22158.988} C_VEL
LIN {X 0,Y 216.901,Z 947.417,A -85,B 0,C 180,E1 22164.844,E2 22164.844} C_VEL
LIN {X 0,Y 190.629,Z 971.335,A -85,B 0,C 180,E1 22173.072,E2 22173.072} C_VEL
LIN {X 0,Y 166.656,Z 991.08,A -85,B 0,C 180,E1 22185.115,E2 22185.115} C_VEL
LIN {X 0,Y 151.114,Z 1004.238,A -85,B 0,C 180,E1 22199.937,E2 22199.937} C_VEL
LIN {X 0,Y 145.561,Z 1010.102,A -85,B 0,C 180,E1 22211.818,E2 22211.818} C_VEL
LIN {X 0,Y 143.86,Z 1013.04,A -85,B 0,C 180,E1 22223.96,E2 22223.96} C_VEL
LIN {X 0,Y 144.163,Z 1013.427,A -85,B 0,C 180,E1 22230.001,E2 22230.001} C_VEL
LIN {X 0,Y 144.252,Z 1011.943,A -85,B 0,C 180,E1 22242.119,E2 22242.119} C_VEL
LIN {X 0,Y 149.298,Z 1005.934,A -85,B 0,C 180,E1 22257.154,E2 22257.154} C_VEL
LIN {X 0,Y 163.289,Z 993.802,A -85,B 0,C 180,E1 22272.492,E2 22272.492} C_VEL
LIN {X 0,Y 182.969,Z 977.806,A -85,B 0,C 180,E1 22283.788,E2 22283.788} C_VEL
LIN {X 0,Y 209.861,Z 954.287,A -85,B 0,C 180,E1 22293.231,E2 22293.231} C_VEL
LIN {X 0,Y 238.127,Z 925.573,A -85,B 0,C 180,E1 22299.885,E2 22299.885} C_VEL
LIN {X 0,Y 265.143,Z 892.384,A -85,B 0,C 180,E1 22304.504,E2 22304.504} C_VEL
LIN {X 0,Y 268.441,Z 887.757,A -85,B 0,C 180,E1 22304.979,E2 22304.979} C_VEL
LIN {X 0,Y 269.617,Z 879.759,A -85,B 0,C 180,E1 22309.478,E2 22309.478} C_VEL
LIN {X 0,Y 269.804,Z 873.758,A -85,B 0,C 180,E1 22315.164,E2 22315.164} C_VEL
LIN {X 0,Y 269.881,Z 871.533,A -85,B 0,C 180,E1 22319.992,E2 22319.992} C_VEL
LIN {X 0,Y 268.743,Z 874.212,A -85,B 0,C 180,E1 22326.461,E2 22326.461} C_VEL
LIN {X 0,Y 267.002,Z 881.987,A -85,B 0,C 180,E1 22333.1,E2 22333.1} C_VEL
LIN {X 0,Y 265.121,Z 888.662,A -85,B 0,C 180,E1 22336.581,E2 22336.581} C_VEL
LIN {X 0,Y 237.955,Z 921.244,A -85,B 0,C 180,E1 22341.473,E2 22341.473} C_VEL
LIN {X 0,Y 210.473,Z 948.241,A -85,B 0,C 180,E1 22348.098,E2 22348.098} C_VEL
LIN {X 0,Y 184.946,Z 969.714,A -85,B 0,C 180,E1 22357.145,E2 22357.145} C_VEL
LIN {X 0,Y 169.231,Z 981.749,A -85,B 0,C 180,E1 22365.417,E2 22365.417} C_VEL
LIN {X 0,Y 158.665,Z 987.512,A -85,B 0,C 180,E1 22369.873,E2 22369.873} C_VEL
LIN {X 0,Y 148.808,Z 992.361,A -85,B 0,C 180,E1 22374.987,E2 22374.987} C_VEL
LIN {X 0,Y 138.806,Z 1000.031,A -85,B 0,C 180,E1 22390.898,E2 22390.898} C_VEL
LIN {X 0,Y 136.184,Z 1002.61,A -85,B 0,C 180,E1 22403.615,E2 22403.615} C_VEL
LIN {X 0,Y 136.216,Z 1002.892,A -85,B 0,C 180,E1 22410.466,E2 22410.466} C_VEL
LIN {X 0,Y 136.97,Z 1001.623,A -85,B 0,C 180,E1 22422.771,E2 22422.771} C_VEL
LIN {X 0,Y 143.504,Z 996.168,A -85,B 0,C 180,E1 22438.344,E2 22438.344} C_VEL
LIN {X 0,Y 157.283,Z 986.367,A -85,B 0,C 180,E1 22452.364,E2 22452.364} C_VEL
LIN {X 0,Y 180.847,Z 969.396,A -85,B 0,C 180,E1 22465.101,E2 22465.101} C_VEL
LIN {X 0,Y 207.912,Z 947.404,A -85,B 0,C 180,E1 22474.106,E2 22474.106} C_VEL
LIN {X 0,Y 236.729,Z 919.593,A -85,B 0,C 180,E1 22480.626,E2 22480.626} C_VEL
LIN {X 0,Y 260.553,Z 891.536,A -85,B 0,C 180,E1 22484.83,E2 22484.83} C_VEL
LIN {X 0,Y 262.936,Z 882.831,A -85,B 0,C 180,E1 22490.953,E2 22490.953} C_VEL
LIN {X 0,Y 264.433,Z 878.48,A -85,B 0,C 180,E1 22496.726,E2 22496.726} C_VEL
LIN {X 0,Y 265.119,Z 877.563,A -85,B 0,C 180,E1 22500.008,E2 22500.008} C_VEL
LIN {X 0,Y 264.897,Z 881.302,A -85,B 0,C 180,E1 22506.571,E2 22506.571} C_VEL
LIN {X 0,Y 263.914,Z 889.382,A -85,B 0,C 180,E1 22512.765,E2 22512.765} C_VEL
LIN {X 0,Y 263.162,Z 891.722,A -85,B 0,C 180,E1 22513.766,E2 22513.766} C_VEL
LIN {X 0,Y 236.067,Z 924.364,A -85,B 0,C 180,E1 22518.103,E2 22518.103} C_VEL
LIN {X 0,Y 208.97,Z 951.323,A -85,B 0,C 180,E1 22523.989,E2 22523.989} C_VEL
LIN {X 0,Y 182.372,Z 974.072,A -85,B 0,C 180,E1 22532.405,E2 22532.405} C_VEL
LIN {X 0,Y 158.859,Z 992.248,A -85,B 0,C 180,E1 22544.373,E2 22544.373} C_VEL
LIN {X 0,Y 144.069,Z 1003.929,A -85,B 0,C 180,E1 22558.301,E2 22558.301} C_VEL
LIN {X 0,Y 137.898,Z 1009.799,A -85,B 0,C 180,E1 22570.769,E2 22570.769} C_VEL
LIN {X 0,Y 135.946,Z 1012.741,A -85,B 0,C 180,E1 22583.607,E2 22583.607} C_VEL
LIN {X 0,Y 136.248,Z 1013.13,A -85,B 0,C 180,E1 22590.001,E2 22590.001} C_VEL
LIN {X 0,Y 136.444,Z 1011.643,A -85,B 0,C 180,E1 22602.824,E2 22602.824} C_VEL
LIN {X 0,Y 142.076,Z 1005.628,A -85,B 0,C 180,E1 22618.658,E2 22618.658} C_VEL
LIN {X 0,Y 156.261,Z 994.295,A -85,B 0,C 180,E1 22633.773,E2 22633.773} C_VEL
LIN {X 0,Y 178.218,Z 977.498,A -85,B 0,C 180,E1 22645.929,E2 22645.929} C_VEL
LIN {X 0,Y 206.191,Z 954.046,A -85,B 0,C 180,E1 22655.266,E2 22655.266} C_VEL
LIN {X 0,Y 235.018,Z 925.739,A -85,B 0,C 180,E1 22661.677,E2 22661.677} C_VEL
LIN {X 0,Y 262.455,Z 892.957,A -85,B 0,C 180,E1 22666.122,E2 22666.122} C_VEL
LIN {X 0,Y 264.001,Z 889.631,A -85,B 0,C 180,E1 22667.158,E2 22667.158} C_VEL
LIN {X 0,Y 264.729,Z 883.255,A -85,B 0,C 180,E1 22671.773,E2 22671.773} C_VEL
LIN {X 0,Y 265.095,Z 879.064,A -85,B 0,C 180,E1 22676.718,E2 22676.718} C_VEL
LIN {X 0,Y 265.14,Z 877.863,A -85,B 0,C 180,E1 22679.992,E2 22679.992} C_VEL
LIN {X 0,Y 263.792,Z 880.675,A -85,B 0,C 180,E1 22686.583,E2 22686.583} C_VEL
LIN {X 0,Y 262.009,Z 887.071,A -85,B 0,C 180,E1 22692.275,E2 22692.275} C_VEL
LIN {X 0,Y 260.505,Z 892.024,A -85,B 0,C 180,E1 22695.263,E2 22695.263} C_VEL
LIN {X 0,Y 233.55,Z 923.121,A -85,B 0,C 180,E1 22699.943,E2 22699.943} C_VEL
LIN {X 0,Y 206.182,Z 949.024,A -85,B 0,C 180,E1 22706.264,E2 22706.264} C_VEL
LIN {X 0,Y 178.518,Z 971.199,A -85,B 0,C 180,E1 22715.754,E2 22715.754} C_VEL
LIN {X 0,Y 155.49,Z 987.666,A -85,B 0,C 180,E1 22728.906,E2 22728.906} C_VEL
LIN {X 0,Y 148.808,Z 992.361,A -85,B 0,C 180,E1 22734.987,E2 22734.987} C_VEL
LIN {X 0,Y 139.969,Z 996.356,A -85,B 0,C 180,E1 22740.788,E2 22740.788} C_VEL
LIN {X 0,Y 132.227,Z 999.49,A -85,B 0,C 180,E1 22747.317,E2 22747.317} C_VEL
LIN {X 0,Y 128.293,Z 1002.908,A -85,B 0,C 180,E1 22763.221,E2 22763.221} C_VEL
LIN {X 0,Y 128.396,Z 1003.206,A -85,B 0,C 180,E1 22769.999,E2 22769.999} C_VEL
LIN {X 0,Y 129.193,Z 1001.922,A -85,B 0,C 180,E1 22783.554,E2 22783.554} C_VEL
LIN {X 0,Y 136.433,Z 996.473,A -85,B 0,C 180,E1 22799.959,E2 22799.959} C_VEL
LIN {X 0,Y 153.252,Z 985.408,A -85,B 0,C 180,E1 22815.698,E2 22815.698} C_VEL
LIN {X 0,Y 176.519,Z 969.542,A -85,B 0,C 180,E1 22827.361,E2 22827.361} C_VEL
LIN {X 0,Y 204.502,Z 947.71,A -85,B 0,C 180,E1 22836.15,E2 22836.15} C_VEL
LIN {X 0,Y 234.17,Z 919.899,A -85,B 0,C 180,E1 22842.494,E2 22842.494} C_VEL
LIN {X 0,Y 254.901,Z 896.557,A -85,B 0,C 180,E1 22845.835,E2 22845.835} C_VEL
LIN {X 0,Y 256.845,Z 891.823,A -85,B 0,C 180,E1 22848.645,E2 22848.645} C_VEL
LIN {X 0,Y 258.749,Z 886.163,A -85,B 0,C 180,E1 22854.128,E2 22854.128} C_VEL
LIN {X 0,Y 260.186,Z 883.77,A -85,B 0,C 180,E1 22860.008,E2 22860.008} C_VEL
LIN {X 0,Y 259.743,Z 887.618,A -85,B 0,C 180,E1 22866.702,E2 22866.702} C_VEL
LIN {X 0,Y 258.637,Z 894.826,A -85,B 0,C 180,E1 22872.279,E2 22872.279} C_VEL
LIN {X 0,Y 230.792,Z 927.126,A -85,B 0,C 180,E1 22876.715,E2 22876.715} C_VEL
LIN {X 0,Y 200.837,Z 955.367,A -85,B 0,C 180,E1 22883.117,E2 22883.117} C_VEL
LIN {X 0,Y 172.901,Z 977.754,A -85,B 0,C 180,E1 22892.154,E2 22892.154} C_VEL
LIN {X 0,Y 148.2,Z 995.548,A -85,B 0,C 180,E1 22905.668,E2 22905.668} C_VEL
LIN {X 0,Y 133.079,Z 1006.929,A -85,B 0,C 180,E1 22922.931,E2 22922.931} C_VEL
LIN {X 0,Y 128.62,Z 1011.329,A -85,B 0,C 180,E1 22936.384,E2 22936.384} C_VEL
LIN {X 0,Y 128.331,Z 1012.833,A -85,B 0,C 180,E1 22950.001,E2 22950.001} C_VEL
LIN {X 0,Y 128.621,Z 1011.342,A -85,B 0,C 180,E1 22963.618,E2 22963.618} C_VEL
LIN {X 0,Y 134.948,Z 1005.322,A -85,B 0,C 180,E1 22980.325,E2 22980.325} C_VEL
LIN {X 0,Y 151.237,Z 993.376,A -85,B 0,C 180,E1 22996.539,E2 22996.539} C_VEL
LIN {X 0,Y 175.173,Z 976.065,A -85,B 0,C 180,E1 23008.752,E2 23008.752} C_VEL
LIN {X 0,Y 203.261,Z 953.383,A -85,B 0,C 180,E1 23017.489,E2 23017.489} C_VEL
LIN {X 0,Y 232.958,Z 925.007,A -85,B 0,C 180,E1 23023.666,E2 23023.666} C_VEL
LIN {X 0,Y 258.736,Z 894.971,A -85,B 0,C 180,E1 23027.697,E2 23027.697} C_VEL
LIN {X 0,Y 259.753,Z 887.874,A -85,B 0,C 180,E1 23033.298,E2 23033.298} C_VEL
LIN {X 0,Y 260.093,Z 885.279,A -85,B 0,C 180,E1 23036.655,E2 23036.655} C_VEL
LIN {X 0,Y 260.204,Z 884.044,A -85,B 0,C 180,E1 23039.992,E2 23039.992} C_VEL
LIN {X 0,Y 258.828,Z 886.452,A -85,B 0,C 180,E1 23046.028,E2 23046.028} C_VEL
LIN {X 0,Y 256.413,Z 893.642,A -85,B 0,C 180,E1 23052.547,E2 23052.547} C_VEL
LIN {X 0,Y 254.868,Z 896.804,A -85,B 0,C 180,E1 23054.059,E2 23054.059} C_VEL
LIN {X 0,Y 227.721,Z 926.574,A -85,B 0,C 180,E1 23058.652,E2 23058.652} C_VEL
LIN {X 0,Y 200.233,Z 951.322,A -85,B 0,C 180,E1 23064.85,E2 23064.85} C_VEL
LIN {X 0,Y 173.21,Z 971.964,A -85,B 0,C 180,E1 23073.856,E2 23073.856} C_VEL
LIN {X 0,Y 149.462,Z 987.97,A -85,B 0,C 180,E1 23086.858,E2 23086.858} C_VEL
LIN {X 0,Y 134.398,Z 998.031,A -85,B 0,C 180,E1 23103.215,E2 23103.215} C_VEL
LIN {X 0,Y 132.227,Z 999.49,A -85,B 0,C 180,E1 23107.317,E2 23107.317} C_VEL
LIN {X 0,Y 127.574,Z 1001.27,A -85,B 0,C 180,E1 23112.678,E2 23112.678} C_VEL
LIN {X 0,Y 120.577,Z 1003.012,A -85,B 0,C 180,E1 23121.257,E2 23121.257} C_VEL
LIN {X 0,Y 120.441,Z 1003.142,A -85,B 0,C 180,E1 23122.302,E2 23122.302} C_VEL
LIN {X 0,Y 120.486,Z 1003.502,A -85,B 0,C 180,E1 23129.999,E2 23129.999} C_VEL
LIN {X 0,Y 121.452,Z 1002.222,A -85,B 0,C 180,E1 23144.436,E2 23144.436} C_VEL
LIN {X 0,Y 129.5,Z 996.776,A -85,B 0,C 180,E1 23161.743,E2 23161.743} C_VEL
LIN {X 0,Y 147.676,Z 985.714,A -85,B 0,C 180,E1 23177.961,E2 23177.961} C_VEL
LIN {X 0,Y 171.538,Z 970.366,A -85,B 0,C 180,E1 23189.378,E2 23189.378} C_VEL
LIN {X 0,Y 201.867,Z 947.574,A -85,B 0,C 180,E1 23198.394,E2 23198.394} C_VEL
LIN {X 0,Y 231.866,Z 920.205,A -85,B 0,C 180,E1 23204.4,E2 23204.4} C_VEL
LIN {X 0,Y 250.338,Z 900.164,A -85,B 0,C 180,E1 23207.226,E2 23207.226} C_VEL
LIN {X 0,Y 252.55,Z 894.655,A -85,B 0,C 180,E1 23211.39,E2 23211.39} C_VEL
LIN {X 0,Y 254.299,Z 890.896,A -85,B 0,C 180,E1 23216.595,E2 23216.595} C_VEL
LIN {X 0,Y 255.146,Z 889.902,A -85,B 0,C 180,E1 23220.008,E2 23220.008} C_VEL
LIN {X 0,Y 254.774,Z 892.442,A -85,B 0,C 180,E1 23225.122,E2 23225.122} C_VEL
LIN {X 0,Y 253.527,Z 898.605,A -85,B 0,C 180,E1 23230.776,E2 23230.776} C_VEL
LIN {X 0,Y 251.697,Z 901.17,A -85,B 0,C 180,E1 23231.306,E2 23231.306} C_VEL
LIN {X 0,Y 224.274,Z 931.01,A -85,B 0,C 180,E1 23235.468,E2 23235.468} C_VEL
LIN {X 0,Y 195.306,Z 957.015,A -85,B 0,C 180,E1 23241.523,E2 23241.523} C_VEL
LIN {X 0,Y 168.152,Z 977.787,A -85,B 0,C 180,E1 23249.969,E2 23249.969} C_VEL
LIN {X 0,Y 141.931,Z 995.526,A -85,B 0,C 180,E1 23263.679,E2 23263.679} C_VEL
LIN {X 0,Y 125.857,Z 1006.622,A -85,B 0,C 180,E1 23281.237,E2 23281.237} C_VEL
LIN {X 0,Y 120.819,Z 1011.027,A -85,B 0,C 180,E1 23295.486,E2 23295.486} C_VEL
LIN {X 0,Y 120.43,Z 1012.537,A -85,B 0,C 180,E1 23310.001,E2 23310.001} C_VEL
LIN {X 0,Y 120.82,Z 1011.041,A -85,B 0,C 180,E1 23324.516,E2 23324.516} C_VEL
LIN {X 0,Y 127.945,Z 1005.016,A -85,B 0,C 180,E1 23342.178,E2 23342.178} C_VEL
LIN {X 0,Y 145.694,Z 993.068,A -85,B 0,C 180,E1 23358.891,E2 23358.891} C_VEL
LIN {X 0,Y 170.305,Z 976.307,A -85,B 0,C 180,E1 23370.838,E2 23370.838} C_VEL
LIN {X 0,Y 199.79,Z 953.481,A -85,B 0,C 180,E1 23379.555,E2 23379.555} C_VEL
LIN {X 0,Y 230.763,Z 924.741,A -85,B 0,C 180,E1 23385.604,E2 23385.604} C_VEL
LIN {X 0,Y 253.031,Z 899.796,A -85,B 0,C 180,E1 23388.835,E2 23388.835} C_VEL
LIN {X 0,Y 254.213,Z 895.907,A -85,B 0,C 180,E1 23391.43,E2 23391.43} C_VEL
LIN {X 0,Y 255.02,Z 891.462,A -85,B 0,C 180,E1 23396.589,E2 23396.589} C_VEL
LIN {X 0,Y 255.167,Z 890.172,A -85,B 0,C 180,E1 23399.992,E2 23399.992} C_VEL
LIN {X 0,Y 253.823,Z 892.119,A -85,B 0,C 180,E1 23405.296,E2 23405.296} C_VEL
LIN {X 0,Y 251.291,Z 898.419,A -85,B 0,C 180,E1 23411.599,E2 23411.599} C_VEL
LIN {X 0,Y 250.273,Z 900.483,A -85,B 0,C 180,E1 23412.703,E2 23412.703} C_VEL
LIN {X 0,Y 220.716,Z 931.284,A -85,B 0,C 180,E1 23417.546,E2 23417.546} C_VEL
LIN {X 0,Y 189.573,Z 957.448,A -85,B 0,C 180,E1 23424.699,E2 23424.699} C_VEL
LIN {X 0,Y 160.999,Z 977.439,A -85,B 0,C 180,E1 23434.799,E2 23434.799} C_VEL
LIN {X 0,Y 138.168,Z 991.596,A -85,B 0,C 180,E1 23448.889,E2 23448.889} C_VEL
LIN {X 0,Y 124.516,Z 1000.021,A -85,B 0,C 180,E1 23466.589,E2 23466.589} C_VEL
LIN {X 0,Y 120.441,Z 1003.142,A -85,B 0,C 180,E1 23482.302,E2 23482.302} C_VEL
LIN {X 0,Y 117.781,Z 1003.709,A -85,B 0,C 180,E1 23488.455,E2 23488.455} C_VEL
LIN {X 0,Y 112.607,Z 1003.296,A -85,B 0,C 180,E1 23499.279,E2 23499.279} C_VEL
LIN {X 0,Y 117.524,Z 1000.06,A -85,B 0,C 180,E1 23515.659,E2 23515.659} C_VEL
LIN {X 0,Y 132.23,Z 991.802,A -85,B 0,C 180,E1 23533.393,E2 23533.393} C_VEL
LIN {X 0,Y 156.641,Z 977.596,A -85,B 0,C 180,E1 23547.591,E2 23547.591} C_VEL
LIN {X 0,Y 187.898,Z 956.453,A -85,B 0,C 180,E1 23557.919,E2 23557.919} C_VEL
LIN {X 0,Y 219.801,Z 930.082,A -85,B 0,C 180,E1 23564.659,E2 23564.659} C_VEL
LIN {X 0,Y 245.019,Z 904.533,A -85,B 0,C 180,E1 23568.537,E2 23568.537} C_VEL
LIN {X 0,Y 247.406,Z 899.935,A -85,B 0,C 180,E1 23572.143,E2 23572.143} C_VEL
LIN {X 0,Y 248.94,Z 896.872,A -85,B 0,C 180,E1 23576.522,E2 23576.522} C_VEL
LIN {X 0,Y 249.903,Z 895.869,A -85,B 0,C 180,E1 23580.008,E2 23580.008} C_VEL
LIN {X 0,Y 249.378,Z 898.466,A -85,B 0,C 180,E1 23585.233,E2 23585.233} C_VEL
LIN {X 0,Y 248.387,Z 902.905,A -85,B 0,C 180,E1 23589.519,E2 23589.519} C_VEL
LIN {X 0,Y 220.03,Z 932.808,A -85,B 0,C 180,E1 23593.784,E2 23593.784} C_VEL
LIN {X 0,Y 189.315,Z 959.158,A -85,B 0,C 180,E1 23599.996,E2 23599.996} C_VEL
LIN {X 0,Y 160.771,Z 979.688,A -85,B 0,C 180,E1 23608.735,E2 23608.735} C_VEL
LIN {X 0,Y 134.454,Z 996.332,A -85,B 0,C 180,E1 23622.519,E2 23622.519} C_VEL
LIN {X 0,Y 118.754,Z 1006.315,A -85,B 0,C 180,E1 23639.338,E2 23639.338} C_VEL
LIN {X 0,Y 113.049,Z 1010.725,A -85,B 0,C 180,E1 23654.464,E2 23654.464} C_VEL
LIN {X 0,Y 112.509,Z 1012.24,A -85,B 0,C 180,E1 23670.001,E2 23670.001} C_VEL
LIN {X 0,Y 113.05,Z 1010.74,A -85,B 0,C 180,E1 23685.539,E2 23685.539} C_VEL
LIN {X 0,Y 121.032,Z 1004.752,A -85,B 0,C 180,E1 23704.147,E2 23704.147} C_VEL
LIN {X 0,Y 140.4,Z 992.759,A -85,B 0,C 180,E1 23721.432,E2 23721.432} C_VEL
LIN {X 0,Y 165.934,Z 976.362,A -85,B 0,C 180,E1 23733.14,E2 23733.14} C_VEL
LIN {X 0,Y 197.192,Z 953.066,A -85,B 0,C 180,E1 23741.829,E2 23741.829} C_VEL
LIN {X 0,Y 228.689,Z 924.611,A -85,B 0,C 180,E1 23747.572,E2 23747.572} C_VEL
LIN {X 0,Y 248.48,Z 903.119,A -85,B 0,C 180,E1 23750.395,E2 23750.395} C_VEL
LIN {X 0,Y 249.677,Z 897.462,A -85,B 0,C 180,E1 23756.515,E2 23756.515} C_VEL
LIN {X 0,Y 249.922,Z 896.115,A -85,B 0,C 180,E1 23759.992,E2 23759.992} C_VEL
LIN {X 0,Y 248.482,Z 898.023,A -85,B 0,C 180,E1 23765.235,E2 23765.235} C_VEL
LIN {X 0,Y 245.872,Z 903.698,A -85,B 0,C 180,E1 23771.084,E2 23771.084} C_VEL
LIN {X 0,Y 217.487,Z 932.391,A -85,B 0,C 180,E1 23775.677,E2 23775.677} C_VEL
LIN {X 0,Y 186.25,Z 957.799,A -85,B 0,C 180,E1 23782.442,E2 23782.442} C_VEL
LIN {X 0,Y 156.404,Z 977.795,A -85,B 0,C 180,E1 23792.39,E2 23792.39} C_VEL
LIN {X 0,Y 132.142,Z 991.901,A -85,B 0,C 180,E1 23806.567,E2 23806.567} C_VEL
LIN {X 0,Y 117.522,Z 1000.113,A -85,B 0,C 180,E1 23824.343,E2 23824.343} C_VEL
LIN {X 0,Y 112.55,Z 1003.503,A -85,B 0,C 180,E1 23842.267,E2 23842.267} C_VEL
LIN {X 0,Y 112.575,Z 1003.799,A -85,B 0,C 180,E1 23849.999,E2 23849.999} C_VEL
LIN {X 0,Y 112.607,Z 1003.296,A -85,B 0,C 180,E1 23859.279,E2 23859.279} C_VEL
LIN {X 0,Y 111.214,Z 1002.598,A -85,B 0,C 180,E1 23865.931,E2 23865.931} C_VEL
LIN {X 0,Y 110.202,Z 1000.424,A -85,B 0,C 180,E1 23877.267,E2 23877.267} C_VEL
LIN {X 0,Y 126.427,Z 992.109,A -85,B 0,C 180,E1 23895.934,E2 23895.934} C_VEL
LIN {X 0,Y 152.885,Z 977.646,A -85,B 0,C 180,E1 23910.339,E2 23910.339} C_VEL
LIN {X 0,Y 184.391,Z 957.205,A -85,B 0,C 180,E1 23920.12,E2 23920.12} C_VEL
LIN {X 0,Y 216.216,Z 931.854,A -85,B 0,C 180,E1 23926.445,E2 23926.445} C_VEL
LIN {X 0,Y 239.808,Z 908.869,A -85,B 0,C 180,E1 23929.918,E2 23929.918} C_VEL
LIN {X 0,Y 241.359,Z 906.497,A -85,B 0,C 180,E1 23931.44,E2 23931.44} C_VEL
LIN {X 0,Y 243.56,Z 902.806,A -85,B 0,C 180,E1 23936.445,E2 23936.445} C_VEL
LIN {X 0,Y 244.593,Z 901.764,A -85,B 0,C 180,E1 23940.009,E2 23940.009} C_VEL
LIN {X 0,Y 243.692,Z 905.233,A -85,B 0,C 180,E1 23946.235,E2 23946.235} C_VEL
LIN {X 0,Y 242.449,Z 908.008,A -85,B 0,C 180,E1 23948.402,E2 23948.402} C_VEL
LIN {X 0,Y 211.847,Z 938.249,A -85,B 0,C 180,E1 23952.69,E2 23952.69} C_VEL
LIN {X 0,Y 180.287,Z 963.585,A -85,B 0,C 180,E1 23959.13,E2 23959.13} C_VEL
LIN {X 0,Y 150.696,Z 983.364,A -85,B 0,C 180,E1 23968.464,E2 23968.464} C_VEL
LIN {X 0,Y 124.558,Z 998.622,A -85,B 0,C 180,E1 23983.171,E2 23983.171} C_VEL
LIN {X 0,Y 109.619,Z 1007.308,A -85,B 0,C 180,E1 24001.092,E2 24001.092} C_VEL
LIN {X 0,Y 104.32,Z 1011.545,A -85,B 0,C 180,E1 24021.656,E2 24021.656} C_VEL
LIN {X 0,Y 104.585,Z 1011.943,A -85,B 0,C 180,E1 24030.002,E2 24030.002} C_VEL
LIN {X 0,Y 105.328,Z 1010.439,A -85,B 0,C 180,E1 24046.71,E2 24046.71} C_VEL
LIN {X 0,Y 113.724,Z 1004.823,A -85,B 0,C 180,E1 24065.602,E2 24065.602} C_VEL
LIN {X 0,Y 133.074,Z 993.832,A -85,B 0,C 180,E1 24082.794,E2 24082.794} C_VEL
LIN {X 0,Y 162.745,Z 975.785,A -85,B 0,C 180,E1 24095.882,E2 24095.882} C_VEL
LIN {X 0,Y 194.545,Z 952.955,A -85,B 0,C 180,E1 24104.081,E2 24104.081} C_VEL
LIN {X 0,Y 227.067,Z 924.307,A -85,B 0,C 180,E1 24109.591,E2 24109.591} C_VEL
LIN {X 0,Y 242.515,Z 908.173,A -85,B 0,C 180,E1 24111.579,E2 24111.579} C_VEL
LIN {X 0,Y 243.704,Z 905.452,A -85,B 0,C 180,E1 24113.752,E2 24113.752} C_VEL
LIN {X 0,Y 244.621,Z 902,A -85,B 0,C 180,E1 24119.991,E2 24119.991} C_VEL
LIN {X 0,Y 243.154,Z 903.693,A -85,B 0,C 180,E1 24124.925,E2 24124.925} C_VEL
LIN {X 0,Y 240.964,Z 907.64,A -85,B 0,C 180,E1 24129.479,E2 24129.479} C_VEL
LIN {X 0,Y 238.842,Z 910.138,A -85,B 0,C 180,E1 24130.123,E2 24130.123} C_VEL
LIN {X 0,Y 209.38,Z 937.849,A -85,B 0,C 180,E1 24134.624,E2 24134.624} C_VEL
LIN {X 0,Y 178.695,Z 961.242,A -85,B 0,C 180,E1 24141.244,E2 24141.244} C_VEL
LIN {X 0,Y 150.22,Z 979.191,A -85,B 0,C 180,E1 24150.6,E2 24150.6} C_VEL
LIN {X 0,Y 126.343,Z 992.206,A -85,B 0,C 180,E1 24164.023,E2 24164.023} C_VEL
LIN {X 0,Y 110.305,Z 1000.415,A -85,B 0,C 180,E1 24182.529,E2 24182.529} C_VEL
LIN {X 0,Y 104.7,Z 1003.8,A -85,B 0,C 180,E1 24201.684,E2 24201.684} C_VEL
LIN {X 0,Y 104.682,Z 1004.095,A -85,B 0,C 180,E1 24209.998,E2 24209.998} C_VEL
LIN {X 0,Y 106.039,Z 1002.822,A -85,B 0,C 180,E1 24226.591,E2 24226.591} C_VEL
LIN {X 0,Y 110.202,Z 1000.424,A -85,B 0,C 180,E1 24237.267,E2 24237.267} C_VEL
LIN {X 0,Y 111.986,Z 997.956,A -85,B 0,C 180,E1 24246.171,E2 24246.171} C_VEL
LIN {X 0,Y 115.85,Z 994.762,A -85,B 0,C 180,E1 24254.671,E2 24254.671} C_VEL
LIN {X 0,Y 142.249,Z 981.562,A -85,B 0,C 180,E1 24270.439,E2 24270.439} C_VEL
LIN {X 0,Y 173.269,Z 963.201,A -85,B 0,C 180,E1 24280.473,E2 24280.473} C_VEL
LIN {X 0,Y 205.338,Z 939.78,A -85,B 0,C 180,E1 24287.097,E2 24287.097} C_VEL
LIN {X 0,Y 235.762,Z 912.019,A -85,B 0,C 180,E1 24291.702,E2 24291.702} C_VEL
LIN {X 0,Y 237.917,Z 908.536,A -85,B 0,C 180,E1 24296.361,E2 24296.361} C_VEL
LIN {X 0,Y 239.057,Z 907.468,A -85,B 0,C 180,E1 24300.009,E2 24300.009} C_VEL
LIN {X 0,Y 238.237,Z 910.264,A -85,B 0,C 180,E1 24305.48,E2 24305.48} C_VEL
LIN {X 0,Y 237.308,Z 912.101,A -85,B 0,C 180,E1 24306.959,E2 24306.959} C_VEL
LIN {X 0,Y 206.645,Z 940.967,A -85,B 0,C 180,E1 24311.061,E2 24311.061} C_VEL
LIN {X 0,Y 174.507,Z 965.492,A -85,B 0,C 180,E1 24317.373,E2 24317.373} C_VEL
LIN {X 0,Y 144.089,Z 984.636,A -85,B 0,C 180,E1 24326.727,E2 24326.727} C_VEL
LIN {X 0,Y 116.972,Z 999.37,A -85,B 0,C 180,E1 24341.905,E2 24341.905} C_VEL
LIN {X 0,Y 100.518,Z 1008.276,A -85,B 0,C 180,E1 24363.137,E2 24363.137} C_VEL
LIN {X 0,Y 96.421,Z 1011.245,A -85,B 0,C 180,E1 24380.967,E2 24380.967} C_VEL
LIN {X 0,Y 96.658,Z 1011.646,A -85,B 0,C 180,E1 24390.002,E2 24390.002} C_VEL
LIN {X 0,Y 97.635,Z 1010.136,A -85,B 0,C 180,E1 24408.07,E2 24408.07} C_VEL
LIN {X 0,Y 106.976,Z 1004.62,A -85,B 0,C 180,E1 24427.906,E2 24427.906} C_VEL
LIN {X 0,Y 128.258,Z 993.524,A -85,B 0,C 180,E1 24445.728,E2 24445.728} C_VEL
LIN {X 0,Y 159.653,Z 975.405,A -85,B 0,C 180,E1 24458.628,E2 24458.628} C_VEL
LIN {X 0,Y 192.981,Z 952.229,A -85,B 0,C 180,E1 24466.53,E2 24466.53} C_VEL
LIN {X 0,Y 225.734,Z 924.003,A -85,B 0,C 180,E1 24471.631,E2 24471.631} C_VEL
LIN {X 0,Y 237.924,Z 911.549,A -85,B 0,C 180,E1 24473.279,E2 24473.279} C_VEL
LIN {X 0,Y 238.647,Z 909.179,A -85,B 0,C 180,E1 24476.354,E2 24476.354} C_VEL
LIN {X 0,Y 239.084,Z 907.684,A -85,B 0,C 180,E1 24479.991,E2 24479.991} C_VEL
LIN {X 0,Y 237.413,Z 909.534,A -85,B 0,C 180,E1 24485.044,E2 24485.044} C_VEL
LIN {X 0,Y 236.003,Z 911.894,A -85,B 0,C 180,E1 24487.95,E2 24487.95} C_VEL
LIN {X 0,Y 233.336,Z 914.706,A -85,B 0,C 180,E1 24488.73,E2 24488.73} C_VEL
LIN {X 0,Y 202.311,Z 942.398,A -85,B 0,C 180,E1 24493.362,E2 24493.362} C_VEL
LIN {X 0,Y 170.281,Z 965.311,A -85,B 0,C 180,E1 24500.207,E2 24500.207} C_VEL
LIN {X 0,Y 137.632,Z 984.127,A -85,B 0,C 180,E1 24511.505,E2 24511.505} C_VEL
LIN {X 0,Y 112.945,Z 996.243,A -85,B 0,C 180,E1 24527.91,E2 24527.91} C_VEL
LIN {X 0,Y 101.685,Z 1001.536,A -85,B 0,C 180,E1 24543.466,E2 24543.466} C_VEL
LIN {X 0,Y 96.833,Z 1004.098,A -85,B 0,C 180,E1 24561.003,E2 24561.003} C_VEL
LIN {X 0,Y 96.768,Z 1004.392,A -85,B 0,C 180,E1 24569.998,E2 24569.998} C_VEL
LIN {X 0,Y 98.398,Z 1003.123,A -85,B 0,C 180,E1 24587.922,E2 24587.922} C_VEL
LIN {X 0,Y 109.572,Z 997.69,A -85,B 0,C 180,E1 24608.447,E2 24608.447} C_VEL
LIN {X 0,Y 115.85,Z 994.762,A -85,B 0,C 180,E1 24614.671,E2 24614.671} C_VEL
LIN {X 0,Y 121.688,Z 990.945,A -85,B 0,C 180,E1 24622.443,E2 24622.443} C_VEL
LIN {X 0,Y 129.214,Z 986.415,A -85,B 0,C 180,E1 24629.404,E2 24629.404} C_VEL
LIN {X 0,Y 160.562,Z 969.695,A -85,B 0,C 180,E1 24640.557,E2 24640.557} C_VEL
LIN {X 0,Y 193.728,Z 947.716,A -85,B 0,C 180,E1 24647.667,E2 24647.667} C_VEL
LIN {X 0,Y 226.03,Z 920.756,A -85,B 0,C 180,E1 24652.435,E2 24652.435} C_VEL
LIN {X 0,Y 230.617,Z 916.311,A -85,B 0,C 180,E1 24653.104,E2 24653.104} C_VEL
LIN {X 0,Y 232.212,Z 914.221,A -85,B 0,C 180,E1 24656.271,E2 24656.271} C_VEL
LIN {X 0,Y 233.473,Z 913.128,A -85,B 0,C 180,E1 24660.009,E2 24660.009} C_VEL
LIN {X 0,Y 232.606,Z 915.643,A -85,B 0,C 180,E1 24665.17,E2 24665.17} C_VEL
LIN {X 0,Y 224.676,Z 923.498,A -85,B 0,C 180,E1 24666.288,E2 24666.288} C_VEL
LIN {X 0,Y 192.23,Z 951.007,A -85,B 0,C 180,E1 24670.913,E2 24670.913} C_VEL
LIN {X 0,Y 159.103,Z 973.553,A -85,B 0,C 180,E1 24677.896,E2 24677.896} C_VEL
LIN {X 0,Y 127.457,Z 991.236,A -85,B 0,C 180,E1 24689.24,E2 24689.24} C_VEL
LIN {X 0,Y 105.386,Z 1002.077,A -85,B 0,C 180,E1 24704.084,E2 24704.084} C_VEL
LIN {X 0,Y 93.334,Z 1007.971,A -85,B 0,C 180,E1 24720.88,E2 24720.88} C_VEL
LIN {X 0,Y 88.534,Z 1010.945,A -85,B 0,C 180,E1 24740.155,E2 24740.155} C_VEL
LIN {X 0,Y 88.733,Z 1011.348,A -85,B 0,C 180,E1 24750.002,E2 24750.002} C_VEL
LIN {X 0,Y 90.011,Z 1009.835,A -85,B 0,C 180,E1 24769.661,E2 24769.661} C_VEL
LIN {X 0,Y 101.325,Z 1003.966,A -85,B 0,C 180,E1 24791.634,E2 24791.634} C_VEL
LIN {X 0,Y 123.783,Z 993.215,A -85,B 0,C 180,E1 24808.897,E2 24808.897} C_VEL
LIN {X 0,Y 157.019,Z 974.968,A -85,B 0,C 180,E1 24821.511,E2 24821.511} C_VEL
LIN {X 0,Y 189.864,Z 952.982,A -85,B 0,C 180,E1 24828.693,E2 24828.693} C_VEL
LIN {X 0,Y 224.688,Z 923.699,A -85,B 0,C 180,E1 24833.698,E2 24833.698} C_VEL
LIN {X 0,Y 231.925,Z 916.634,A -85,B 0,C 180,E1 24834.511,E2 24834.511} C_VEL
LIN {X 0,Y 232.932,Z 914.915,A -85,B 0,C 180,E1 24836.265,E2 24836.265} C_VEL
LIN {X 0,Y 233.504,Z 913.338,A -85,B 0,C 180,E1 24839.991,E2 24839.991} C_VEL
LIN {X 0,Y 231.406,Z 915.449,A -85,B 0,C 180,E1 24845.408,E2 24845.408} C_VEL
LIN {X 0,Y 230.727,Z 916.395,A -85,B 0,C 180,E1 24846.705,E2 24846.705} C_VEL
LIN {X 0,Y 202.376,Z 941.336,A -85,B 0,C 180,E1 24850.806,E2 24850.806} C_VEL
LIN {X 0,Y 166.94,Z 966.029,A -85,B 0,C 180,E1 24857.762,E2 24857.762} C_VEL
LIN {X 0,Y 133.537,Z 984.433,A -85,B 0,C 180,E1 24868.509,E2 24868.509} C_VEL
LIN {X 0,Y 107.067,Z 996.547,A -85,B 0,C 180,E1 24885,E2 24885} C_VEL
LIN {X 0,Y 94.563,Z 1001.836,A -85,B 0,C 180,E1 24901.29,E2 24901.29} C_VEL
LIN {X 0,Y 88.991,Z 1004.396,A -85,B 0,C 180,E1 24920.202,E2 24920.202} C_VEL
LIN {X 0,Y 88.869,Z 1004.688,A -85,B 0,C 180,E1 24929.998,E2 24929.998} C_VEL
LIN {X 0,Y 90.819,Z 1003.423,A -85,B 0,C 180,E1 24949.475,E2 24949.475} C_VEL
LIN {X 0,Y 103.337,Z 997.995,A -85,B 0,C 180,E1 24971.247,E2 24971.247} C_VEL
LIN {X 0,Y 128.194,Z 986.912,A -85,B 0,C 180,E1 24988.9,E2 24988.9} C_VEL
LIN {X 0,Y 129.214,Z 986.415,A -85,B 0,C 180,E1 24989.404,E2 24989.404} C_VEL
LIN {X 0,Y 138.231,Z 981.25,A -85,B 0,C 180,E1 24995.47,E2 24995.47} C_VEL
LIN {X 0,Y 148.278,Z 975.389,A -85,B 0,C 180,E1 25000.74,E2 25000.74} C_VEL
LIN {X 0,Y 182.284,Z 954.918,A -85,B 0,C 180,E1 25008.382,E2 25008.382} C_VEL
LIN {X 0,Y 215.68,Z 929.426,A -85,B 0,C 180,E1 25013.357,E2 25013.357} C_VEL
LIN {X 0,Y 225.484,Z 920.657,A -85,B 0,C 180,E1 25014.774,E2 25014.774} C_VEL
LIN {X 0,Y 227.647,Z 918.566,A -85,B 0,C 180,E1 25020.009,E2 25020.009} C_VEL
LIN {X 0,Y 227.064,Z 920.148,A -85,B 0,C 180,E1 25023.832,E2 25023.832} C_VEL
LIN {X 0,Y 194.871,Z 947.636,A -85,B 0,C 180,E1 25027.862,E2 25027.862} C_VEL
LIN {X 0,Y 160.919,Z 970.767,A -85,B 0,C 180,E1 25034.056,E2 25034.056} C_VEL
LIN {X 0,Y 126.959,Z 989.344,A -85,B 0,C 180,E1 25044.481,E2 25044.481} C_VEL
LIN {X 0,Y 99.838,Z 1001.768,A -85,B 0,C 180,E1 25060.69,E2 25060.69} C_VEL
LIN {X 0,Y 83.382,Z 1008.961,A -85,B 0,C 180,E1 25085.262,E2 25085.262} C_VEL
LIN {X 0,Y 80.799,Z 1011.051,A -85,B 0,C 180,E1 25110.002,E2 25110.002} C_VEL
LIN {X 0,Y 83.385,Z 1008.982,A -85,B 0,C 180,E1 25134.742,E2 25134.742} C_VEL
LIN {X 0,Y 99.843,Z 1001.813,A -85,B 0,C 180,E1 25159.311,E2 25159.311} C_VEL
LIN {X 0,Y 129.04,Z 988.426,A -85,B 0,C 180,E1 25176.401,E2 25176.401} C_VEL
LIN {X 0,Y 165.242,Z 968.284,A -85,B 0,C 180,E1 25186.867,E2 25186.867} C_VEL
LIN {X 0,Y 200.501,Z 943.527,A -85,B 0,C 180,E1 25192.921,E2 25192.921} C_VEL
LIN {X 0,Y 227.022,Z 920.399,A -85,B 0,C 180,E1 25196.167,E2 25196.167} C_VEL
LIN {X 0,Y 227.681,Z 918.756,A -85,B 0,C 180,E1 25199.991,E2 25199.991} C_VEL
LIN {X 0,Y 225.597,Z 920.784,A -85,B 0,C 180,E1 25205.194,E2 25205.194} C_VEL
LIN {X 0,Y 195.642,Z 945.608,A -85,B 0,C 180,E1 25209.34,E2 25209.34} C_VEL
LIN {X 0,Y 164.641,Z 966.332,A -85,B 0,C 180,E1 25215.066,E2 25215.066} C_VEL
LIN {X 0,Y 129.846,Z 984.738,A -85,B 0,C 180,E1 25225.348,E2 25225.348} C_VEL
LIN {X 0,Y 101.473,Z 996.851,A -85,B 0,C 180,E1 25241.748,E2 25241.748} C_VEL
LIN {X 0,Y 86.221,Z 1002.578,A -85,B 0,C 180,E1 25261.339,E2 25261.339} C_VEL
LIN {X 0,Y 81.154,Z 1004.695,A -85,B 0,C 180,E1 25279.245,E2 25279.245} C_VEL
LIN {X 0,Y 80.952,Z 1004.985,A -85,B 0,C 180,E1 25289.998,E2 25289.998} C_VEL
LIN {X 0,Y 83.309,Z 1003.724,A -85,B 0,C 180,E1 25311.312,E2 25311.312} C_VEL
LIN {X 0,Y 97.211,Z 998.368,A -85,B 0,C 180,E1 25334.21,E2 25334.21} C_VEL
LIN {X 0,Y 124.169,Z 987.22,A -85,B 0,C 180,E1 25352.132,E2 25352.132} C_VEL
LIN {X 0,Y 148.278,Z 975.389,A -85,B 0,C 180,E1 25360.74,E2 25360.74} C_VEL
LIN {X 0,Y 159.1,Z 968.931,A -85,B 0,C 180,E1 25365.314,E2 25365.314} C_VEL
LIN {X 0,Y 170.569,Z 961.749,A -85,B 0,C 180,E1 25369.187,E2 25369.187} C_VEL
LIN {X 0,Y 203.572,Z 938.914,A -85,B 0,C 180,E1 25374.135,E2 25374.135} C_VEL
LIN {X 0,Y 219.985,Z 925.375,A -85,B 0,C 180,E1 25376.064,E2 25376.064} C_VEL
LIN {X 0,Y 221.805,Z 923.962,A -85,B 0,C 180,E1 25380.009,E2 25380.009} C_VEL
LIN {X 0,Y 221.393,Z 924.768,A -85,B 0,C 180,E1 25382.169,E2 25382.169} C_VEL
LIN {X 0,Y 186.663,Z 952.701,A -85,B 0,C 180,E1 25386.476,E2 25386.476} C_VEL
LIN {X 0,Y 151.402,Z 974.926,A -85,B 0,C 180,E1 25392.833,E2 25392.833} C_VEL
LIN {X 0,Y 116.098,Z 992.525,A -85,B 0,C 180,E1 25404.095,E2 25404.095} C_VEL
LIN {X 0,Y 86.107,Z 1004.777,A -85,B 0,C 180,E1 25425.306,E2 25425.306} C_VEL
LIN {X 0,Y 75.019,Z 1009.213,A -85,B 0,C 180,E1 25446.196,E2 25446.196} C_VEL
LIN {X 0,Y 72.862,Z 1010.753,A -85,B 0,C 180,E1 25470.002,E2 25470.002} C_VEL
LIN {X 0,Y 75.022,Z 1009.23,A -85,B 0,C 180,E1 25493.808,E2 25493.808} C_VEL
LIN {X 0,Y 90.537,Z 1003.036,A -85,B 0,C 180,E1 25519.427,E2 25519.427} C_VEL
LIN {X 0,Y 118.434,Z 991.508,A -85,B 0,C 180,E1 25536.932,E2 25536.932} C_VEL
LIN {X 0,Y 151.417,Z 975.03,A -85,B 0,C 180,E1 25547.151,E2 25547.151} C_VEL
LIN {X 0,Y 188.481,Z 951.528,A -85,B 0,C 180,E1 25553.779,E2 25553.779} C_VEL
LIN {X 0,Y 220.283,Z 925.976,A -85,B 0,C 180,E1 25557.558,E2 25557.558} C_VEL
LIN {X 0,Y 221.373,Z 924.956,A -85,B 0,C 180,E1 25557.93,E2 25557.93} C_VEL
LIN {X 0,Y 221.839,Z 924.142,A -85,B 0,C 180,E1 25559.991,E2 25559.991} C_VEL
LIN {X 0,Y 219.47,Z 926.024,A -85,B 0,C 180,E1 25563.946,E2 25563.946} C_VEL
LIN {X 0,Y 185.443,Z 952.313,A -85,B 0,C 180,E1 25568.309,E2 25568.309} C_VEL
LIN {X 0,Y 152.036,Z 972.604,A -85,B 0,C 180,E1 25574.612,E2 25574.612} C_VEL
LIN {X 0,Y 117.558,Z 988.925,A -85,B 0,C 180,E1 25585.632,E2 25585.632} C_VEL
LIN {X 0,Y 87.604,Z 1000.153,A -85,B 0,C 180,E1 25606.262,E2 25606.262} C_VEL
LIN {X 0,Y 75.904,Z 1004.051,A -85,B 0,C 180,E1 25626.485,E2 25626.485} C_VEL
LIN {X 0,Y 73.053,Z 1005.281,A -85,B 0,C 180,E1 25649.998,E2 25649.998} C_VEL
LIN {X 0,Y 75.902,Z 1004.024,A -85,B 0,C 180,E1 25673.511,E2 25673.511} C_VEL
LIN {X 0,Y 94.014,Z 997.853,A -85,B 0,C 180,E1 25699.931,E2 25699.931} C_VEL
LIN {X 0,Y 123.566,Z 986.234,A -85,B 0,C 180,E1 25716.776,E2 25716.776} C_VEL
LIN {X 0,Y 155.904,Z 970.309,A -85,B 0,C 180,E1 25726.203,E2 25726.203} C_VEL
LIN {X 0,Y 170.569,Z 961.749,A -85,B 0,C 180,E1 25729.187,E2 25729.187} C_VEL
LIN {X 0,Y 182.444,Z 953.941,A -85,B 0,C 180,E1 25732.539,E2 25732.539} C_VEL
LIN {X 0,Y 194.488,Z 945.462,A -85,B 0,C 180,E1 25735.434,E2 25735.434} C_VEL
LIN {X 0,Y 213.468,Z 930.835,A -85,B 0,C 180,E1 25737.549,E2 25737.549} C_VEL
LIN {X 0,Y 215.011,Z 929.576,A -85,B 0,C 180,E1 25738.734,E2 25738.734} C_VEL
LIN {X 0,Y 215.612,Z 929.286,A -85,B 0,C 180,E1 25740.526,E2 25740.526} C_VEL
LIN {X 0,Y 182.229,Z 954.841,A -85,B 0,C 180,E1 25744.421,E2 25744.421} C_VEL
LIN {X 0,Y 146.274,Z 976.465,A -85,B 0,C 180,E1 25750.478,E2 25750.478} C_VEL
LIN {X 0,Y 109.878,Z 993.493,A -85,B 0,C 180,E1 25761.549,E2 25761.549} C_VEL
LIN {X 0,Y 80.484,Z 1004.469,A -85,B 0,C 180,E1 25781.197,E2 25781.197} C_VEL
LIN {X 0,Y 67.667,Z 1008.925,A -85,B 0,C 180,E1 25803.564,E2 25803.564} C_VEL
LIN {X 0,Y 64.922,Z 1010.456,A -85,B 0,C 180,E1 25830.003,E2 25830.003} C_VEL
LIN {X 0,Y 67.705,Z 1008.928,A -85,B 0,C 180,E1 25856.571,E2 25856.571} C_VEL
LIN {X 0,Y 85.025,Z 1002.866,A -85,B 0,C 180,E1 25883.262,E2 25883.262} C_VEL
LIN {X 0,Y 115.452,Z 991.2,A -85,B 0,C 180,E1 25900.701,E2 25900.701} C_VEL
LIN {X 0,Y 149.794,Z 974.721,A -85,B 0,C 180,E1 25910.239,E2 25910.239} C_VEL
LIN {X 0,Y 187.767,Z 951.221,A -85,B 0,C 180,E1 25916.276,E2 25916.276} C_VEL
LIN {X 0,Y 215.642,Z 929.463,A -85,B 0,C 180,E1 25919.466,E2 25919.466} C_VEL
LIN {X 0,Y 214.45,Z 930.225,A -85,B 0,C 180,E1 25921.866,E2 25921.866} C_VEL
LIN {X 0,Y 210.318,Z 933.677,A -85,B 0,C 180,E1 25922.714,E2 25922.714} C_VEL
LIN {X 0,Y 173.776,Z 959.501,A -85,B 0,C 180,E1 25927.32,E2 25927.32} C_VEL
LIN {X 0,Y 136.948,Z 979.46,A -85,B 0,C 180,E1 25934.667,E2 25934.667} C_VEL
LIN {X 0,Y 102.357,Z 993.725,A -85,B 0,C 180,E1 25947.432,E2 25947.432} C_VEL
LIN {X 0,Y 74.26,Z 1002.742,A -85,B 0,C 180,E1 25972.287,E2 25972.287} C_VEL
LIN {X 0,Y 65.564,Z 1005.292,A -85,B 0,C 180,E1 25996.645,E2 25996.645} C_VEL
LIN {X 0,Y 65.131,Z 1005.578,A -85,B 0,C 180,E1 26009.997,E2 26009.997} C_VEL
LIN {X 0,Y 70.453,Z 1003.712,A -85,B 0,C 180,E1 26040.797,E2 26040.797} C_VEL
LIN {X 0,Y 91.5,Z 997.388,A -85,B 0,C 180,E1 26065.826,E2 26065.826} C_VEL
LIN {X 0,Y 123.801,Z 985.245,A -85,B 0,C 180,E1 26081.405,E2 26081.405} C_VEL
LIN {X 0,Y 162.965,Z 965.799,A -85,B 0,C 180,E1 26090.8,E2 26090.8} C_VEL
LIN {X 0,Y 194.488,Z 945.462,A -85,B 0,C 180,E1 26095.434,E2 26095.434} C_VEL
LIN {X 0,Y 195.272,Z 944.885,A -85,B 0,C 180,E1 26096.549,E2 26096.549} C_VEL
LIN {X 0,Y 191.018,Z 947.929,A -85,B 0,C 180,E1 26098.865,E2 26098.865} C_VEL
LIN {X 0,Y 179.363,Z 956.102,A -85,B 0,C 180,E1 26101.93,E2 26101.93} C_VEL
LIN {X 0,Y 174.95,Z 959.013,A -85,B 0,C 180,E1 26102.643,E2 26102.643} C_VEL
LIN {X 0,Y 137.856,Z 979.722,A -85,B 0,C 180,E1 26108.715,E2 26108.715} C_VEL
LIN {X 0,Y 100.718,Z 995.567,A -85,B 0,C 180,E1 26120.028,E2 26120.028} C_VEL
LIN {X 0,Y 70.167,Z 1005.658,A -85,B 0,C 180,E1 26142.336,E2 26142.336} C_VEL
LIN {X 0,Y 57.265,Z 1009.745,A -85,B 0,C 180,E1 26174.672,E2 26174.672} C_VEL
LIN {X 0,Y 56.977,Z 1010.158,A -85,B 0,C 180,E1 26190.003,E2 26190.003} C_VEL
LIN {X 0,Y 60.571,Z 1008.624,A -85,B 0,C 180,E1 26219.999,E2 26219.999} C_VEL
LIN {X 0,Y 80.376,Z 1002.558,A -85,B 0,C 180,E1 26247.965,E2 26247.965} C_VEL
LIN {X 0,Y 113.854,Z 990.528,A -85,B 0,C 180,E1 26264.965,E2 26264.965} C_VEL
LIN {X 0,Y 148.62,Z 974.414,A -85,B 0,C 180,E1 26273.369,E2 26273.369} C_VEL
LIN {X 0,Y 187.413,Z 950.915,A -85,B 0,C 180,E1 26278.789,E2 26278.789} C_VEL
LIN {X 0,Y 206.385,Z 936.8,A -85,B 0,C 180,E1 26280.854,E2 26280.854} C_VEL
LIN {X 0,Y 171.304,Z 960.744,A -85,B 0,C 180,E1 26284.864,E2 26284.864} C_VEL
LIN {X 0,Y 135.11,Z 979.765,A -85,B 0,C 180,E1 26291.313,E2 26291.313} C_VEL
LIN {X 0,Y 98.868,Z 994.03,A -85,B 0,C 180,E1 26303.236,E2 26303.236} C_VEL
LIN {X 0,Y 68.049,Z 1003.045,A -85,B 0,C 180,E1 26328.122,E2 26328.122} C_VEL
LIN {X 0,Y 57.85,Z 1005.59,A -85,B 0,C 180,E1 26354.825,E2 26354.825} C_VEL
LIN {X 0,Y 57.216,Z 1005.875,A -85,B 0,C 180,E1 26369.997,E2 26369.997} C_VEL
LIN {X 0,Y 61.553,Z 1004.625,A -85,B 0,C 180,E1 26399.467,E2 26399.467} C_VEL
LIN {X 0,Y 81.437,Z 999.315,A -85,B 0,C 180,E1 26426.135,E2 26426.135} C_VEL
LIN {X 0,Y 114.778,Z 988.142,A -85,B 0,C 180,E1 26443.009,E2 26443.009} C_VEL
LIN {X 0,Y 150.421,Z 972.21,A -85,B 0,C 180,E1 26451.695,E2 26451.695} C_VEL
LIN {X 0,Y 187.913,Z 950.031,A -85,B 0,C 180,E1 26457.135,E2 26457.135} C_VEL
LIN {X 0,Y 206.664,Z 936.395,A -85,B 0,C 180,E1 26459.109,E2 26459.109} C_VEL
LIN {X 0,Y 174.95,Z 959.013,A -85,B 0,C 180,E1 26462.643,E2 26462.643} C_VEL
LIN {X 0,Y 159.868,Z 967.837,A -85,B 0,C 180,E1 26463.23,E2 26463.23} C_VEL
LIN {X 0,Y 144.346,Z 975.766,A -85,B 0,C 180,E1 26463.995,E2 26463.995} C_VEL
LIN {X 0,Y 104.932,Z 992.87,A -85,B 0,C 180,E1 26473.108,E2 26473.108} C_VEL
LIN {X 0,Y 70.759,Z 1003.852,A -85,B 0,C 180,E1 26491.145,E2 26491.145} C_VEL
LIN {X 0,Y 51.782,Z 1008.726,A -85,B 0,C 180,E1 26521.375,E2 26521.375} C_VEL
LIN {X 0,Y 49.03,Z 1009.86,A -85,B 0,C 180,E1 26550.003,E2 26550.003} C_VEL
LIN {X 0,Y 53.704,Z 1008.32,A -85,B 0,C 180,E1 26584.327,E2 26584.327} C_VEL
LIN {X 0,Y 76.332,Z 1002.251,A -85,B 0,C 180,E1 26613.207,E2 26613.207} C_VEL
LIN {X 0,Y 111.822,Z 990.285,A -85,B 0,C 180,E1 26629.016,E2 26629.016} C_VEL
LIN {X 0,Y 147.895,Z 974.106,A -85,B 0,C 180,E1 26636.544,E2 26636.544} C_VEL
LIN {X 0,Y 181.717,Z 954.346,A -85,B 0,C 180,E1 26640.94,E2 26640.94} C_VEL
LIN {X 0,Y 144.068,Z 975.262,A -85,B 0,C 180,E1 26646.017,E2 26646.017} C_VEL
LIN {X 0,Y 106.038,Z 990.952,A -85,B 0,C 180,E1 26654.977,E2 26654.977} C_VEL
LIN {X 0,Y 72.022,Z 1001.063,A -85,B 0,C 180,E1 26672.76,E2 26672.76} C_VEL
